Omron CX-Programmer project 新工程 (CX-Programmer 9.73)

# PLC 新PLC1: CQM1H CPU21

## Global symbols (name address type ; comment)
0.00 BOOL  ; 急停
0.01 BOOL  ; 内线
0.02 BOOL  ; 中线
0.03 BOOL  ; 外线
0.04 BOOL  ; 手动上升
0.05 BOOL  ; 手动下降
0.06 BOOL  ; 储坯/进窑
0.07 BOOL  ; 自动/手动
0.08 BOOL  ; 连锁
0.09 BOOL  ; 笼中进
0.10 BOOL  ; 笼中出
0.11 BOOL  ; 新加线开
0.12 BOOL  ; 棒1#光电
0.13 BOOL  ; 棒2#光电
0.14 BOOL  ; 棒3光电
0.15 BOOL  ; 棒8#光电
100.00 BOOL  ; 棒1#快速速
100.01 BOOL  ; 棒1#慢速
100.02 BOOL  ; 内送砖前3#基速
100.03 BOOL  ; 内送砖前3#慢速
100.04 BOOL  ; 中线送砖前3#
100.05 BOOL  ; 中线送砖前3#慢速
100.06 BOOL  ; 外线送砖前3#正转
100.07 BOOL  ; 外线送砖前3#慢速
100.08 BOOL  ; 内线正转
100.09 BOOL  ; 内线慢速
100.10 BOOL  ; 内线反转
100.12 BOOL  ; 中线正转
100.13 BOOL  ; 中线低速
100.14 BOOL  ; 中线反转
101.00 BOOL  ; 外线正转
101.01 BOOL  ; 外线低速
101.02 BOOL  ; 外线反转
101.04 BOOL  ; 棒2#
101.05 BOOL  ; 棒3#
101.06 BOOL  ; 棒4#
101.07 BOOL  ; 棒7#
101.08 BOOL  ; 棒8#
101.09 BOOL  ; 棍9#正转
101.10 BOOL  ; 棍9#反转
101.11 BOOL  ; 棒10#正转
101.12 BOOL  ; 棒10#反转
101.13 BOOL  ; 棒11#正转
101.14 BOOL  ; 棒11#反转
101.15 BOOL  ; 棒12正转（外线）
102.00 BOOL  ; 棒12反转（外线）
102.01 BOOL  ; 1#补棒正转
102.02 BOOL  ; 1#补棒反转
102.03 BOOL  ; 2#补棒正转
102.04 BOOL  ; 2#补棒反转
102.05 BOOL  ; 1#笼棒正转
102.06 BOOL  ; 1#笼棒棒反转
102.07 BOOL  ; 2#笼棒正转
102.08 BOOL  ; 2#笼棒反转
102.09 BOOL  ; 内线送砖前2#
102.10 BOOL  ; 内送砖前1#
102.11 BOOL  ; 内线送砖
102.12 BOOL  ; 内线步进
102.13 BOOL  ; 内线升降
102.14 BOOL  ; 中线送砖前2#
102.15 BOOL  ; 中线送砖前1#
103.00 BOOL  ; 中线送砖
103.01 BOOL  ; 中线步进
103.02 BOOL  ; 中线升降
103.03 BOOL  ; 外线送砖前2#
103.04 BOOL  ; 外线送砖前1#
103.05 BOOL  ; 外线送砖
103.06 BOOL  ; 吊笼上升
103.07 BOOL  ; 吊笼下降
103.08 BOOL  ; 外线步进
103.09 BOOL  ; 外线升降
104.00 BOOL  ; 1线快拉正转
104.01 BOOL  ; 1线快拉反转
104.02 BOOL  ; 1线快拉慢速
104.03 BOOL  ; 1线送砖前4#基速
104.04 BOOL  ; 1线送砖前4#慢速
104.05 BOOL  ; 1线送砖前3#
104.06 BOOL  ; 1线送砖前2#
104.07 BOOL  ; 1线送砖前1#
104.08 BOOL  ; 1线送砖
104.09 BOOL  ; 1线步进
104.10 BOOL  ; 1线升降
104.11 BOOL  ; 棒5
104.12 BOOL  ; 棒6#
10.00 BOOL  ; 砖已离开补棒1#
10.01 BOOL  ; 棒11#放砖
10.02 BOOL  ; 棒11#放砖
10.03 BOOL  ; 棒9#正转
10.05 BOOL  ; 棒9反储启棒10反
10.06 BOOL  ; 棒10反储启棒11反
11.00 BOOL  ; 吊笼自动上升
11.01 BOOL  ; 吊笼手动上升
11.02 BOOL  ; 吊笼上升定位
11.03 BOOL  ; 吊笼自下
11.04 BOOL  ; 吊笼手下
11.05 BOOL  ; 下降定位
11.07 BOOL  ; 补棒1#有砖
12.00 BOOL  ; 棒12#正转
1.00 BOOL  ; 棒10#光电
1.01 BOOL  ; 棒11#光电
1.02 BOOL  ; 补棒光电
1.03 BOOL  ; 补棒对射
1.04 BOOL  ; 吊笼进口对射
1.05 BOOL  ; 斜射
1.06 BOOL  ; 吊笼定长
1.07 BOOL  ; 吊笼定位
1.08 BOOL  ; 上升层定位
1.09 BOOL  ; 下降层限
1.10 BOOL  ; 上限
1.11 BOOL  ; 下限
1.12 BOOL  ; 内送砖前3#光电
1.13 BOOL  ; 内送砖前2#光电
1.14 BOOL  ; 内送砖前1#光电
1.15 BOOL  ; 内线送砖光电
20.00 BOOL  ; 棒7正转
2.00 BOOL  ; 内线定位光电
2.01 BOOL  ; 内线升降接近
2.02 BOOL  ; 内正限
2.03 BOOL  ; 内正慢
2.04 BOOL  ; 内反慢
2.05 BOOL  ; 内反限
2.06 BOOL  ; 中线1#光电
2.07 BOOL  ; 中线送砖前2#光电
2.08 BOOL  ; 中线送砖前1#光电
2.09 BOOL  ; 中线送砖光电
2.10 BOOL  ; 中线定位光电
2.11 BOOL  ; 中线升降接近
2.12 BOOL  ; 中正限
2.13 BOOL  ; 中正慢
2.14 BOOL  ; 中反慢
2.15 BOOL  ; 中反限
3.00 BOOL  ; 外线送砖前3#光电
3.01 BOOL  ; 外线送砖前2#光电
3.02 BOOL  ; 外线送砖前1#光电
3.03 BOOL  ; 外线送砖光电
3.04 BOOL  ; 外线定位光电
3.05 BOOL  ; 外线升降接近
3.06 BOOL  ; 外正限
3.07 BOOL  ; 外正慢
3.08 BOOL  ; 外反慢
3.09 BOOL  ; 外反限
3.14 BOOL  ; 棒4光电
4.00 BOOL  ; 1线快拉正限
4.01 BOOL  ; 1线快拉正慢
4.02 BOOL  ; 1线快拉反限
4.03 BOOL  ; 1线快拉反慢
4.04 BOOL  ; 1线送砖前4#光电
4.05 BOOL  ; 1线送砖前3#光电
4.06 BOOL  ; 1线送砖前2#光电
4.07 BOOL  ; 1线送砖前1#光电
4.08 BOOL  ; 1线送砖光电
4.09 BOOL  ; 1线定位光电
4.10 BOOL  ; 1线升降接近
4.11 BOOL  ; 棒6光电
CNT005 BOOL  ; 棒12#过砖时间
CNT007 BOOL  ; 棒12#放砖时间
CNT008 BOOL  ; 棒11#放砖时间
CNT009 BOOL  ; 棒10#放砖时间
CNT013 BOOL  ; 棒9#放砖时间
CNT015 BOOL  ; 棒9#过砖时间
CNT021 BOOL  ; 棒8放砖时间
CNT022 BOOL  ; 棒7#过砖时间
CNT024 BOOL  ; 棒7#放砖时间
CNT028 BOOL  ; 棒9#反储时间
CNT030 BOOL  ; 棒10#反储时间
CNT032 BOOL  ; 棒11#反储时间
CNT033 BOOL  ; 棒12#反过时间
CNT035 BOOL  ; 棒12#反储时间
CNT038 BOOL  ; 吊笼上升到位
CNT041 BOOL  ; 下降定位
CNT045 BOOL  ; 补棒1#反储定位
CNT051 BOOL  ; 棒11反储时间
CNT053 BOOL  ; 棒10#放砖时间
CNT102 BOOL  ; 棒6放砖时间
CNT103 BOOL  ; 棒5#过砖时间
CNT105 BOOL  ; 棒5#放砖时间
HR0.01 BOOL  ; 内线上升
HR0.02 BOOL  ; 内线快拉正转
HR0.03 BOOL  ; 内线下降
HR0.04 BOOL  ; 内线快拉反转
HR0.05 BOOL  ; 中线上升
HR0.06 BOOL  ; 中线快拉正转
HR0.07 BOOL  ; 中线下降
HR0.08 BOOL  ; 中线快拉反转
HR0.09 BOOL  ; 外线上升
HR0.10 BOOL  ; 外线快拉正转
HR0.11 BOOL  ; 外线下降
HR0.12 BOOL  ; 外线快拉反转
HR0.13 BOOL  ; 笼棒放砖
HR0.14 BOOL  ; 棒12#过砖
HR0.15 BOOL  ; 棒12#放砖
HR10.00 BOOL  ; 棒12放砖至棒11
HR10.01 BOOL  ; 棒11#放砖
HR10.02 BOOL  ; 棒11放砖至棒10
HR10.03 BOOL  ; 棒10#放砖
HR10.04 BOOL  ; 棒9#中线放砖
HR10.05 BOOL  ; 棒9#过砖
HR10.06 BOOL  ; 棒9放砖至棒8
HR10.07 BOOL  ; 棒8#放砖
HR10.08 BOOL  ; 棒7#过砖
HR10.09 BOOL  ; 棒7#放砖
HR10.10 BOOL  ; 中线储坯下降
HR10.11 BOOL  ; 外线储坯下降
HR10.12 BOOL  ; 棒9#反储
HR10.13 BOOL  ; 棒10#反过
HR10.14 BOOL  ; 棒10#反储
HR10.15 BOOL  ; 棒11#反过
HR11.00 BOOL  ; 棒11#反储
HR11.01 BOOL  ; 棒12#反过
HR11.02 BOOL  ; 棒12#反储
HR11.03 BOOL  ; 笼棒反储定长
HR12.00 BOOL  ; 吊笼上升
HR12.01 BOOL  ; 吊笼下降
HR12.02 BOOL  ; 补棒1#反储定长
HR12.04 BOOL  ; 棒10#反储
HR12.05 BOOL  ; 棒10有砖棒11反储
HR12.06 BOOL  ; 棒12放砖至棒11
HR12.07 BOOL  ; 棒10#放砖
HR13.01 BOOL  ; 1线上升
HR13.02 BOOL  ; 1线快拉正转
HR13.03 BOOL  ; 1线下降
HR13.04 BOOL  ; 1线快拉反转
HR13.08 BOOL  ; 棒7放砖至棒6
HR13.09 BOOL  ; 棒6#放砖
HR13.10 BOOL  ; 棒5#过砖
HR13.11 BOOL  ; 棒5#放砖
TIM000 BOOL  ; 棒1#无砖
TIM001 BOOL  ; 内线快拉正转后
TIM002 BOOL  ; 中线快拉正转
TIM003 BOOL  ; 外线快拉正转
TIM004 BOOL  ; 放砖条件
TIM006 BOOL  ; 外线下降
TIM010 BOOL  ; 棒11砖定位
TIM011 BOOL  ; 棒10砖定位
TIM012 BOOL  ; 中线下降
TIM020 BOOL  ; 棒8#砖定位
TIM023 BOOL  ; 内线下降
TIM025 BOOL  ; 中线储坯下降条件
TIM026 BOOL  ; 外线储坯下降条件
TIM027 BOOL  ; 中线储坯下降
TIM029 BOOL  ; 棒10#反过定位
TIM031 BOOL  ; 棒11#反过定位
TIM034 BOOL  ; 外线储坯下降
TIM036 BOOL  ; 吊笼上升条件
TIM037 BOOL  ; 上升层定位
TIM039 BOOL  ; 吊笼下降条件
TIM040 BOOL  ; 下降层定位
TIM042 BOOL  ; 棒10#放砖条件
TIM043 BOOL  ; 棒11放砖条件
TIM050 BOOL  ; 定位
TIM052 BOOL  ; 棒11砖定位
TIM055 BOOL  ; 棒10#放砖条件
TIM100 BOOL  ; 1线快拉正转后
TIM101 BOOL  ; 棒6#砖定位
TIM104 BOOL  ; 1线下降

## Program 新程序1 (no task)
; 程序使用CX-Programmer 9.75编写，PLC型号为CQM1H CPU21。程序实现了陶瓷厂储坯器系统的控制系统，通过输送带控制坯料输送、升降机调整坯料位置和吊笼实现坯料存储。操作人员通过自动/手动开关选择运行模式，自动和手动模式不能同时启用。 / 设备情况：输送带、升降机、吊笼、急停按钮、连锁开关、光电传感器、限位开关和接近开关等。 / 操作员可以通过自动/手动开关选择运行模式，在自动模式下，运转准备信号和插头连接确认信号确认后点亮自动运转指示灯。若插头连接确认信号为假，检测暂停，自动运转指示灯不点亮，直到插头重新连接。检测流程由放水电磁阀和电机运转继电器控制，通过压力到达信号确保压力达标。 / 输送带控制方面，内线启动按钮启动内线正转输出，需内线送砖光电持续为真。内线输送启动前，确认内线送砖光电信号。中线启动按钮控制中线正转输出，需中线送砖光电信号正常；中线输送启动前，检测中线送砖光电状态。外线启动按钮控制外线正转输出，需外线送砖光电信号有效；外线输送启动前，确保外线送砖光电有效。内线升降输出运行时，需内线升降接近为真以确认位置；内线升降启动时，检查内线升降接近是否到位；内线升降完成时，记录运行状态；内线正转输出此时停止，避免部件掉落。 / 吊笼由吊笼上升输出和吊笼下降输出控制，在自动模式下由运转准备信号和上限信号触发上升，手动模式下由手动上升按钮和手动下降按钮操作。吊笼停止前，检测吊笼进口对射是否正常。吊笼运行时，吊笼进口对射必须为真以检测障碍物，否则停止运行，避免撞击。吊笼定位控制移动，上限信号和下限信号限制移动范围。 / 安全方面，急停按钮按下时，内线正转输出、吊笼上升输出等所有输出立即停止，确保人员和设备安全；系统启动前，检测急停按钮是否复位。若连锁开关为假，内线正转输出、电机运转继电器等主要输出停止运行，防止不安全状态下的操作；输送开始前，确认连锁开关已闭合。不良状态下，操作员按下不良解除按钮可复位系统，恢复初始状态。 / 内线正转输出运行时需持续检测内线送砖光电，中线正转输出需持续检测中线送砖光电，外线正转输出需持续检测外线送砖光电，否则停止运行以防部件堆积。 / 内线升降输出运行时需持续检测内线升降接近，中线升降输出需持续检测中线升降接近，外线升降输出需持续检测外线升降接近，以确保位置正常；中线升降前，验证中线升降接近信号；外线升降开始前，确认外线升降接近正常。

### Section 段1

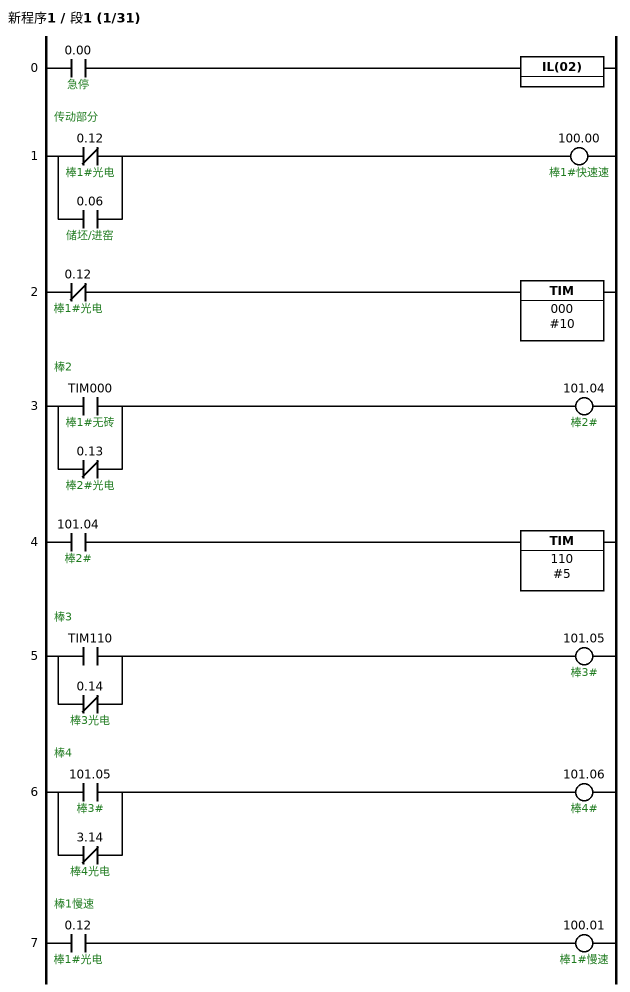
; rung 0
LD 0.00  ; 急停
IL(02)
; rung 1: 传动部分
LDNOT 0.12  ; 棒1#光电
OR 0.06  ; 储坯/进窑
OUT 100.00  ; 棒1#快速速
; rung 2
LDNOT 0.12  ; 棒1#光电
TIM 000 #10
; rung 3: 棒2
LD TIM000  ; 棒1#无砖
ORNOT 0.13  ; 棒2#光电
OUT 101.04  ; 棒2#
; rung 4
LD 101.04  ; 棒2#
TIM 110 #5
; rung 5: 棒3
LD TIM110
ORNOT 0.14  ; 棒3光电
OUT 101.05  ; 棒3#
; rung 6: 棒4
LD 101.05  ; 棒3#
ORNOT 3.14  ; 棒4光电
OUT 101.06  ; 棒4#
; rung 7: 棒1慢速
LD 0.12  ; 棒1#光电
OUT 100.01  ; 棒1#慢速

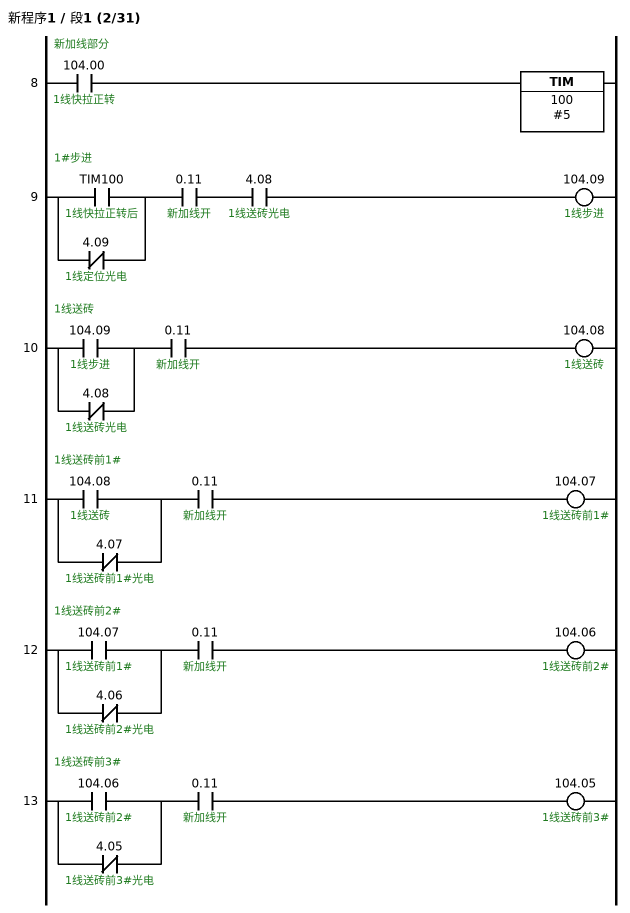
; rung 8: 新加线部分
LD 104.00  ; 1线快拉正转
TIM 100 #5
; rung 9: 1#步进
LD TIM100  ; 1线快拉正转后
ORNOT 4.09  ; 1线定位光电
AND 0.11  ; 新加线开
AND 4.08  ; 1线送砖光电
OUT 104.09  ; 1线步进
; rung 10: 1线送砖
LD 104.09  ; 1线步进
ORNOT 4.08  ; 1线送砖光电
AND 0.11  ; 新加线开
OUT 104.08  ; 1线送砖
; rung 11: 1线送砖前1#
LD 104.08  ; 1线送砖
ORNOT 4.07  ; 1线送砖前1#光电
AND 0.11  ; 新加线开
OUT 104.07  ; 1线送砖前1#
; rung 12: 1线送砖前2#
LD 104.07  ; 1线送砖前1#
ORNOT 4.06  ; 1线送砖前2#光电
AND 0.11  ; 新加线开
OUT 104.06  ; 1线送砖前2#
; rung 13: 1线送砖前3#
LD 104.06  ; 1线送砖前2#
ORNOT 4.05  ; 1线送砖前3#光电
AND 0.11  ; 新加线开
OUT 104.05  ; 1线送砖前3#

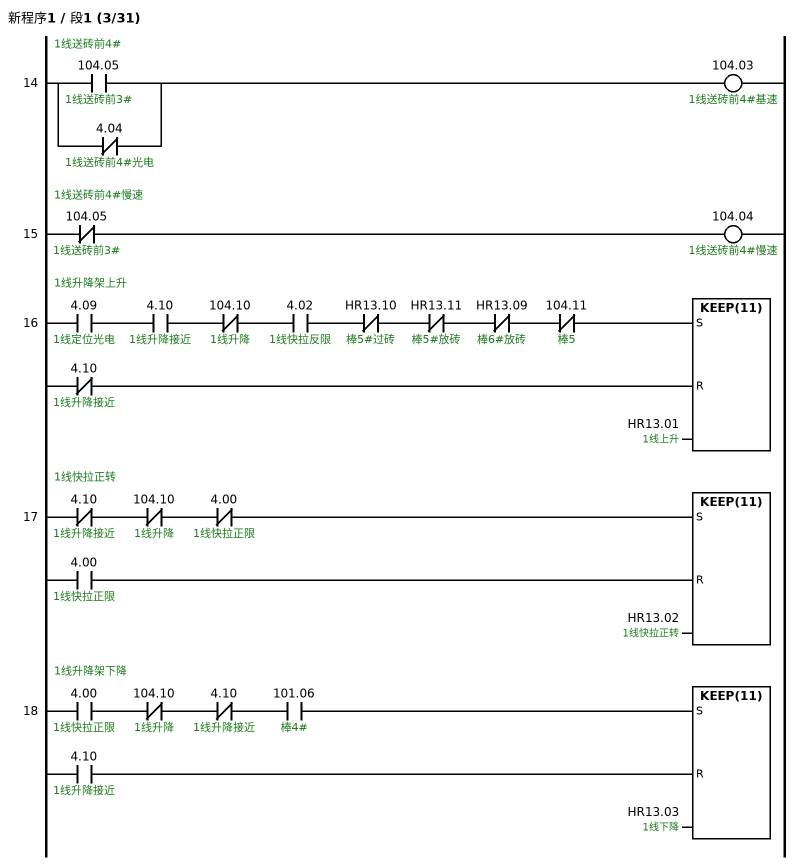
; rung 14: 1线送砖前4#
LD 104.05  ; 1线送砖前3#
ORNOT 4.04  ; 1线送砖前4#光电
OUT 104.03  ; 1线送砖前4#基速
; rung 15: 1线送砖前4#慢速
LDNOT 104.05  ; 1线送砖前3#
OUT 104.04  ; 1线送砖前4#慢速
; rung 16: 1线升降架上升
LD 4.09  ; 1线定位光电
AND 4.10  ; 1线升降接近
ANDNOT 104.10  ; 1线升降
AND 4.02  ; 1线快拉反限
ANDNOT HR13.10  ; 棒5#过砖
ANDNOT HR13.11  ; 棒5#放砖
ANDNOT HR13.09  ; 棒6#放砖
ANDNOT 104.11  ; 棒5
LDNOT 4.10  ; 1线升降接近
KEEP(11) HR13.01  ; 1线上升
; rung 17: 1线快拉正转
LDNOT 4.10  ; 1线升降接近
ANDNOT 104.10  ; 1线升降
ANDNOT 4.00  ; 1线快拉正限
LD 4.00  ; 1线快拉正限
KEEP(11) HR13.02  ; 1线快拉正转
; rung 18: 1线升降架下降
LD 4.00  ; 1线快拉正限
ANDNOT 104.10  ; 1线升降
ANDNOT 4.10  ; 1线升降接近
AND 101.06  ; 棒4#
LD 4.10  ; 1线升降接近
KEEP(11) HR13.03  ; 1线下降

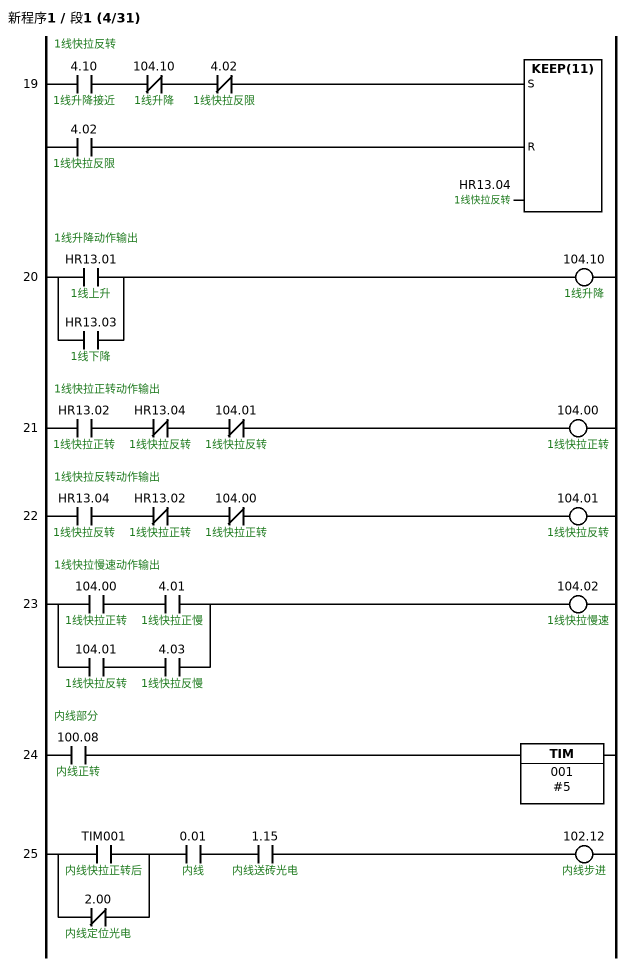
; rung 19: 1线快拉反转
LD 4.10  ; 1线升降接近
ANDNOT 104.10  ; 1线升降
ANDNOT 4.02  ; 1线快拉反限
LD 4.02  ; 1线快拉反限
KEEP(11) HR13.04  ; 1线快拉反转
; rung 20: 1线升降动作输出
LD HR13.01  ; 1线上升
OR HR13.03  ; 1线下降
OUT 104.10  ; 1线升降
; rung 21: 1线快拉正转动作输出
LD HR13.02  ; 1线快拉正转
ANDNOT HR13.04  ; 1线快拉反转
ANDNOT 104.01  ; 1线快拉反转
OUT 104.00  ; 1线快拉正转
; rung 22: 1线快拉反转动作输出
LD HR13.04  ; 1线快拉反转
ANDNOT HR13.02  ; 1线快拉正转
ANDNOT 104.00  ; 1线快拉正转
OUT 104.01  ; 1线快拉反转
; rung 23: 1线快拉慢速动作输出
LD 104.00  ; 1线快拉正转
AND 4.01  ; 1线快拉正慢
LD 104.01  ; 1线快拉反转
AND 4.03  ; 1线快拉反慢
ORLD
OUT 104.02  ; 1线快拉慢速
; rung 24: 内线部分
LD 100.08  ; 内线正转
TIM 001 #5
; rung 25
LD TIM001  ; 内线快拉正转后
ORNOT 2.00  ; 内线定位光电
AND 0.01  ; 内线
AND 1.15  ; 内线送砖光电
OUT 102.12  ; 内线步进

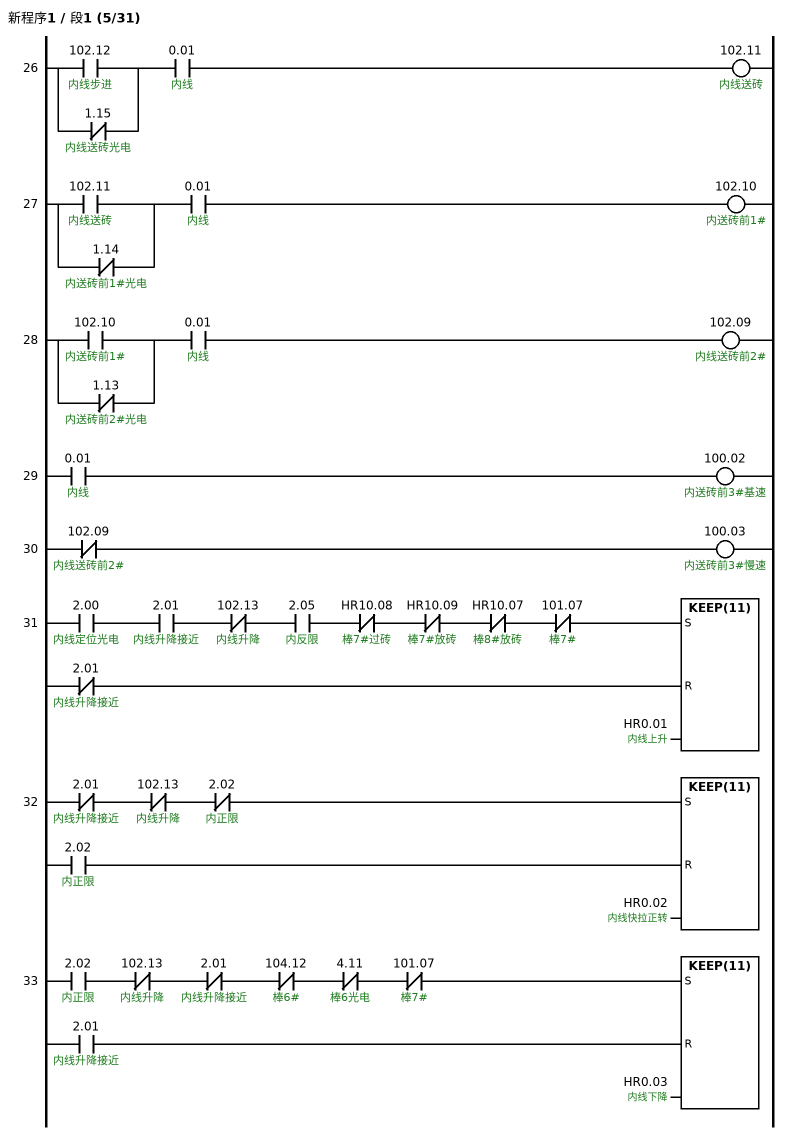
; rung 26
LD 102.12  ; 内线步进
ORNOT 1.15  ; 内线送砖光电
AND 0.01  ; 内线
OUT 102.11  ; 内线送砖
; rung 27
LD 102.11  ; 内线送砖
ORNOT 1.14  ; 内送砖前1#光电
AND 0.01  ; 内线
OUT 102.10  ; 内送砖前1#
; rung 28
LD 102.10  ; 内送砖前1#
ORNOT 1.13  ; 内送砖前2#光电
AND 0.01  ; 内线
OUT 102.09  ; 内线送砖前2#
; rung 29
LD 0.01  ; 内线
OUT 100.02  ; 内送砖前3#基速
; rung 30
LDNOT 102.09  ; 内线送砖前2#
OUT 100.03  ; 内送砖前3#慢速
; rung 31
LD 2.00  ; 内线定位光电
AND 2.01  ; 内线升降接近
ANDNOT 102.13  ; 内线升降
AND 2.05  ; 内反限
ANDNOT HR10.08  ; 棒7#过砖
ANDNOT HR10.09  ; 棒7#放砖
ANDNOT HR10.07  ; 棒8#放砖
ANDNOT 101.07  ; 棒7#
LDNOT 2.01  ; 内线升降接近
KEEP(11) HR0.01  ; 内线上升
; rung 32
LDNOT 2.01  ; 内线升降接近
ANDNOT 102.13  ; 内线升降
ANDNOT 2.02  ; 内正限
LD 2.02  ; 内正限
KEEP(11) HR0.02  ; 内线快拉正转
; rung 33
LD 2.02  ; 内正限
ANDNOT 102.13  ; 内线升降
ANDNOT 2.01  ; 内线升降接近
ANDNOT 104.12  ; 棒6#
ANDNOT 4.11  ; 棒6光电
ANDNOT 101.07  ; 棒7#
LD 2.01  ; 内线升降接近
KEEP(11) HR0.03  ; 内线下降

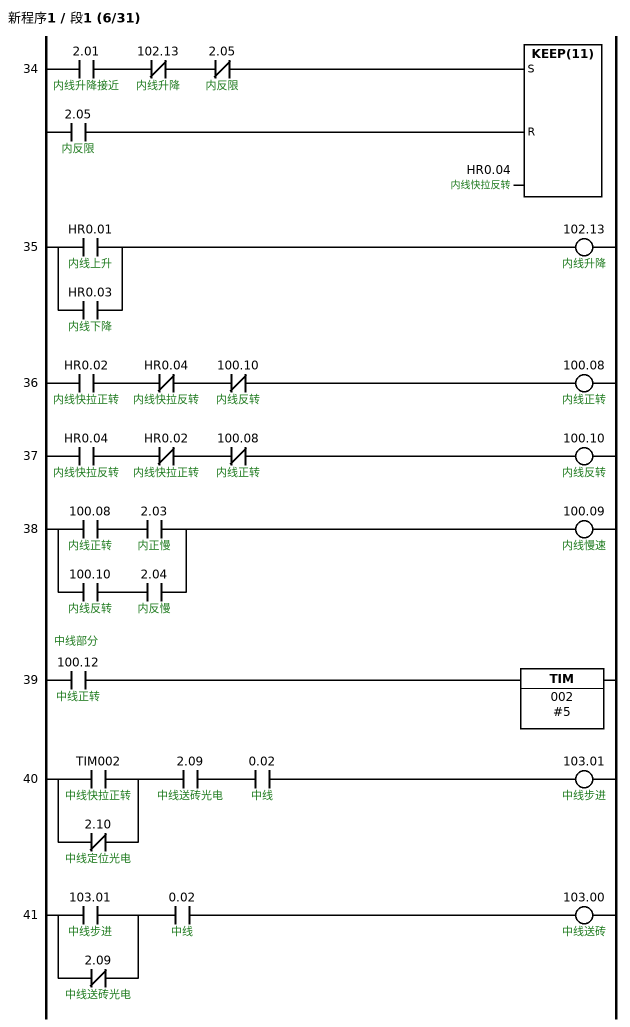
; rung 34
LD 2.01  ; 内线升降接近
ANDNOT 102.13  ; 内线升降
ANDNOT 2.05  ; 内反限
LD 2.05  ; 内反限
KEEP(11) HR0.04  ; 内线快拉反转
; rung 35
LD HR0.01  ; 内线上升
OR HR0.03  ; 内线下降
OUT 102.13  ; 内线升降
; rung 36
LD HR0.02  ; 内线快拉正转
ANDNOT HR0.04  ; 内线快拉反转
ANDNOT 100.10  ; 内线反转
OUT 100.08  ; 内线正转
; rung 37
LD HR0.04  ; 内线快拉反转
ANDNOT HR0.02  ; 内线快拉正转
ANDNOT 100.08  ; 内线正转
OUT 100.10  ; 内线反转
; rung 38
LD 100.08  ; 内线正转
AND 2.03  ; 内正慢
LD 100.10  ; 内线反转
AND 2.04  ; 内反慢
ORLD
OUT 100.09  ; 内线慢速
; rung 39: 中线部分
LD 100.12  ; 中线正转
TIM 002 #5
; rung 40
LD TIM002  ; 中线快拉正转
ORNOT 2.10  ; 中线定位光电
AND 2.09  ; 中线送砖光电
AND 0.02  ; 中线
OUT 103.01  ; 中线步进
; rung 41
LD 103.01  ; 中线步进
ORNOT 2.09  ; 中线送砖光电
AND 0.02  ; 中线
OUT 103.00  ; 中线送砖

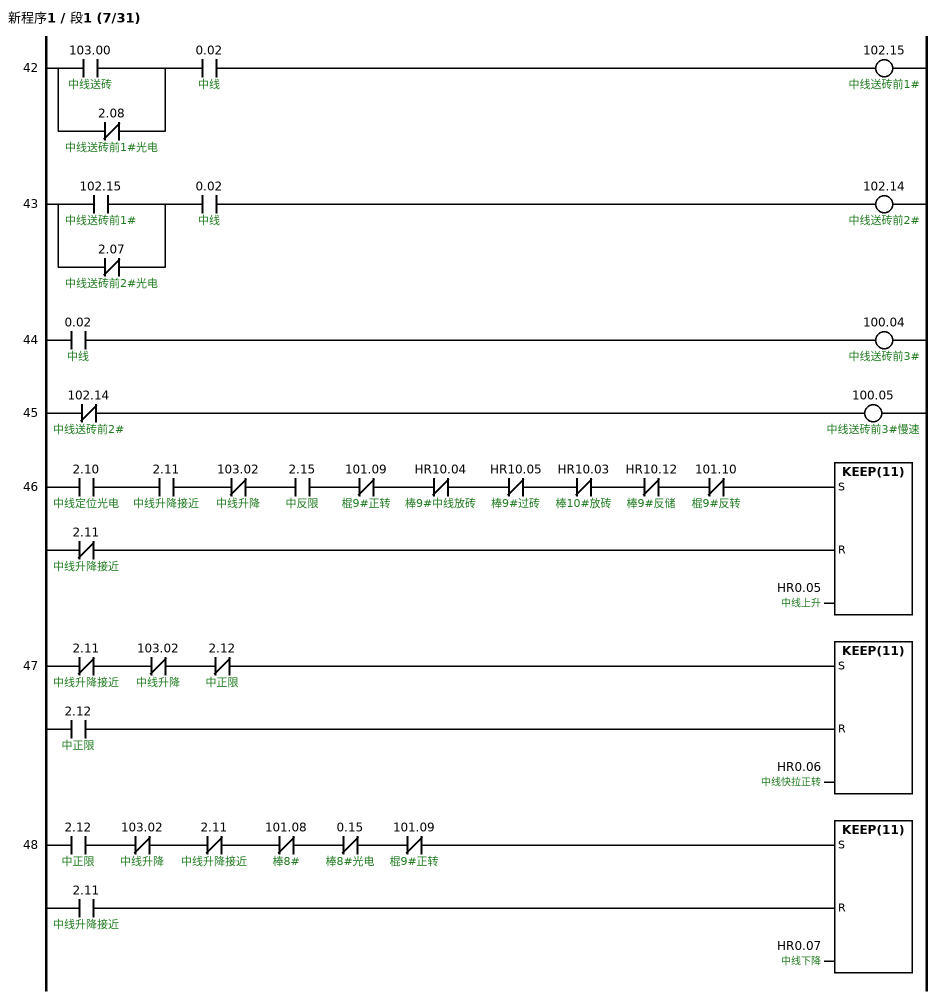
; rung 42
LD 103.00  ; 中线送砖
ORNOT 2.08  ; 中线送砖前1#光电
AND 0.02  ; 中线
OUT 102.15  ; 中线送砖前1#
; rung 43
LD 102.15  ; 中线送砖前1#
ORNOT 2.07  ; 中线送砖前2#光电
AND 0.02  ; 中线
OUT 102.14  ; 中线送砖前2#
; rung 44
LD 0.02  ; 中线
OUT 100.04  ; 中线送砖前3#
; rung 45
LDNOT 102.14  ; 中线送砖前2#
OUT 100.05  ; 中线送砖前3#慢速
; rung 46
LD 2.10  ; 中线定位光电
AND 2.11  ; 中线升降接近
ANDNOT 103.02  ; 中线升降
AND 2.15  ; 中反限
ANDNOT 101.09  ; 棍9#正转
ANDNOT HR10.04  ; 棒9#中线放砖
ANDNOT HR10.05  ; 棒9#过砖
ANDNOT HR10.03  ; 棒10#放砖
ANDNOT HR10.12  ; 棒9#反储
ANDNOT 101.10  ; 棍9#反转
LDNOT 2.11  ; 中线升降接近
KEEP(11) HR0.05  ; 中线上升
; rung 47
LDNOT 2.11  ; 中线升降接近
ANDNOT 103.02  ; 中线升降
ANDNOT 2.12  ; 中正限
LD 2.12  ; 中正限
KEEP(11) HR0.06  ; 中线快拉正转
; rung 48
LD 2.12  ; 中正限
ANDNOT 103.02  ; 中线升降
ANDNOT 2.11  ; 中线升降接近
ANDNOT 101.08  ; 棒8#
ANDNOT 0.15  ; 棒8#光电
ANDNOT 101.09  ; 棍9#正转
LD 2.11  ; 中线升降接近
KEEP(11) HR0.07  ; 中线下降

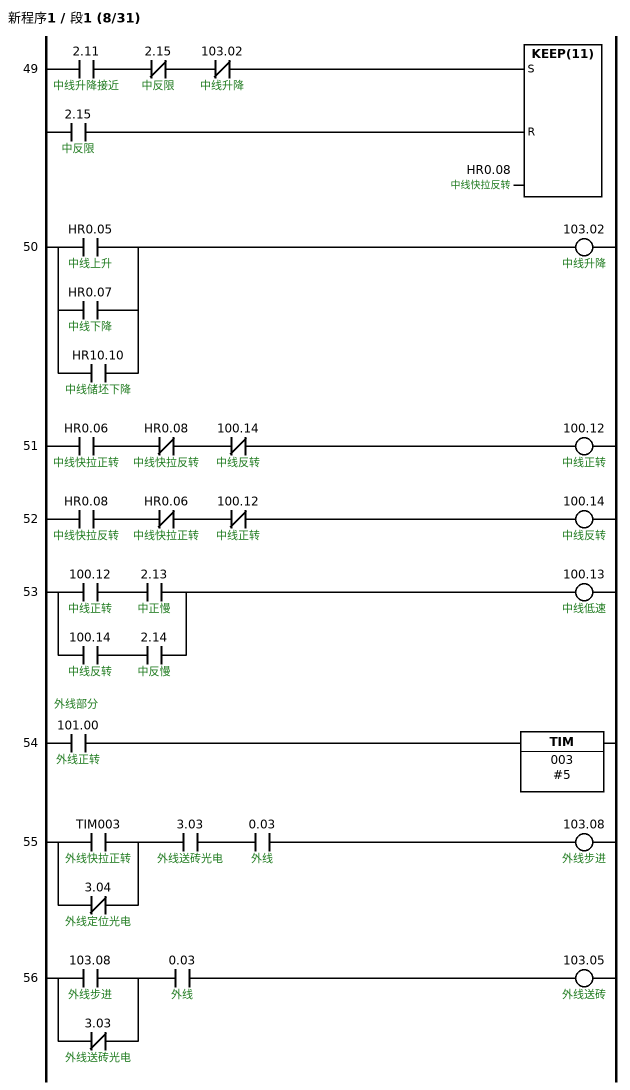
; rung 49
LD 2.11  ; 中线升降接近
ANDNOT 2.15  ; 中反限
ANDNOT 103.02  ; 中线升降
LD 2.15  ; 中反限
KEEP(11) HR0.08  ; 中线快拉反转
; rung 50
LD HR0.05  ; 中线上升
OR HR0.07  ; 中线下降
OR HR10.10  ; 中线储坯下降
OUT 103.02  ; 中线升降
; rung 51
LD HR0.06  ; 中线快拉正转
ANDNOT HR0.08  ; 中线快拉反转
ANDNOT 100.14  ; 中线反转
OUT 100.12  ; 中线正转
; rung 52
LD HR0.08  ; 中线快拉反转
ANDNOT HR0.06  ; 中线快拉正转
ANDNOT 100.12  ; 中线正转
OUT 100.14  ; 中线反转
; rung 53
LD 100.12  ; 中线正转
AND 2.13  ; 中正慢
LD 100.14  ; 中线反转
AND 2.14  ; 中反慢
ORLD
OUT 100.13  ; 中线低速
; rung 54: 外线部分
LD 101.00  ; 外线正转
TIM 003 #5
; rung 55
LD TIM003  ; 外线快拉正转
ORNOT 3.04  ; 外线定位光电
AND 3.03  ; 外线送砖光电
AND 0.03  ; 外线
OUT 103.08  ; 外线步进
; rung 56
LD 103.08  ; 外线步进
ORNOT 3.03  ; 外线送砖光电
AND 0.03  ; 外线
OUT 103.05  ; 外线送砖

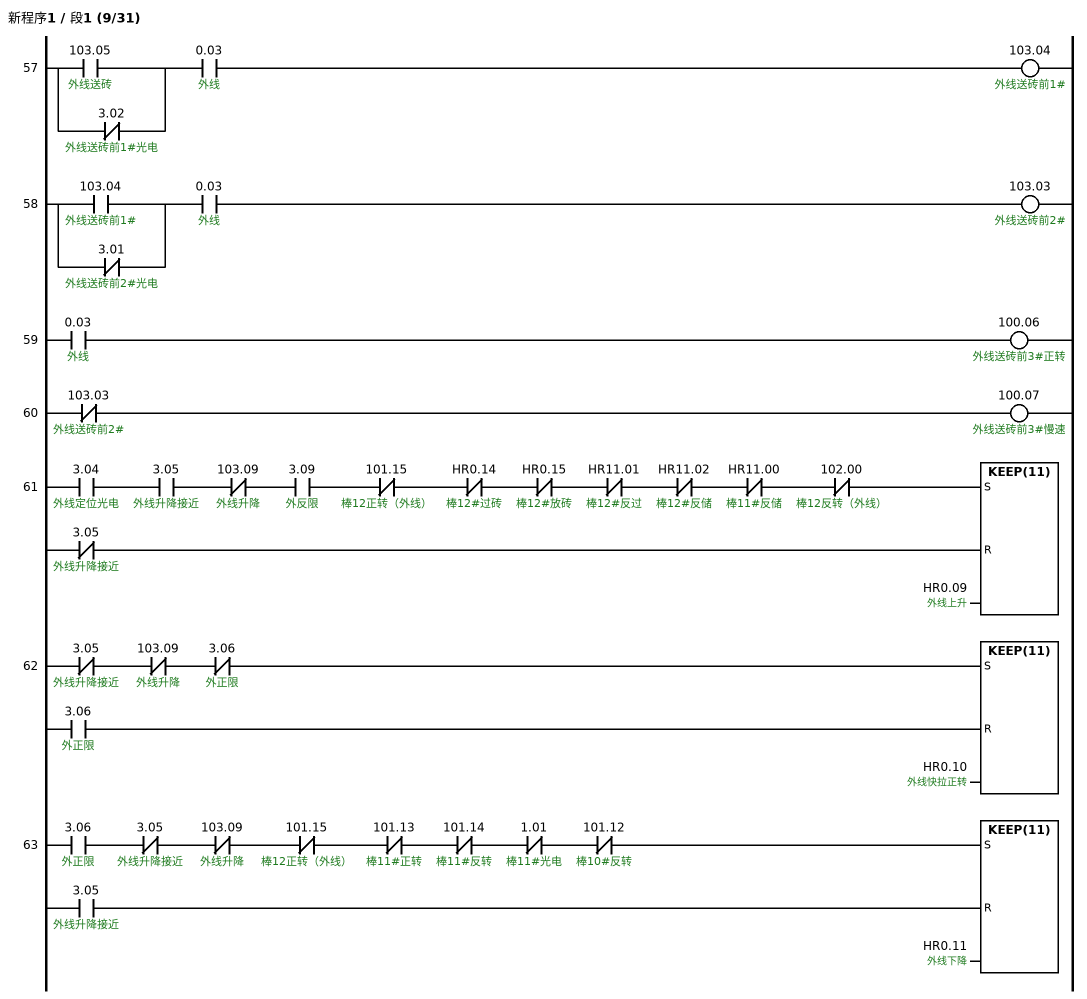
; rung 57
LD 103.05  ; 外线送砖
ORNOT 3.02  ; 外线送砖前1#光电
AND 0.03  ; 外线
OUT 103.04  ; 外线送砖前1#
; rung 58
LD 103.04  ; 外线送砖前1#
ORNOT 3.01  ; 外线送砖前2#光电
AND 0.03  ; 外线
OUT 103.03  ; 外线送砖前2#
; rung 59
LD 0.03  ; 外线
OUT 100.06  ; 外线送砖前3#正转
; rung 60
LDNOT 103.03  ; 外线送砖前2#
OUT 100.07  ; 外线送砖前3#慢速
; rung 61
LD 3.04  ; 外线定位光电
AND 3.05  ; 外线升降接近
ANDNOT 103.09  ; 外线升降
AND 3.09  ; 外反限
ANDNOT 101.15  ; 棒12正转（外线）
ANDNOT HR0.14  ; 棒12#过砖
ANDNOT HR0.15  ; 棒12#放砖
ANDNOT HR11.01  ; 棒12#反过
ANDNOT HR11.02  ; 棒12#反储
ANDNOT HR11.00  ; 棒11#反储
ANDNOT 102.00  ; 棒12反转（外线）
LDNOT 3.05  ; 外线升降接近
KEEP(11) HR0.09  ; 外线上升
; rung 62
LDNOT 3.05  ; 外线升降接近
ANDNOT 103.09  ; 外线升降
ANDNOT 3.06  ; 外正限
LD 3.06  ; 外正限
KEEP(11) HR0.10  ; 外线快拉正转
; rung 63
LD 3.06  ; 外正限
ANDNOT 3.05  ; 外线升降接近
ANDNOT 103.09  ; 外线升降
ANDNOT 101.15  ; 棒12正转（外线）
ANDNOT 101.13  ; 棒11#正转
ANDNOT 101.14  ; 棒11#反转
ANDNOT 1.01  ; 棒11#光电
ANDNOT 101.12  ; 棒10#反转
LD 3.05  ; 外线升降接近
KEEP(11) HR0.11  ; 外线下降

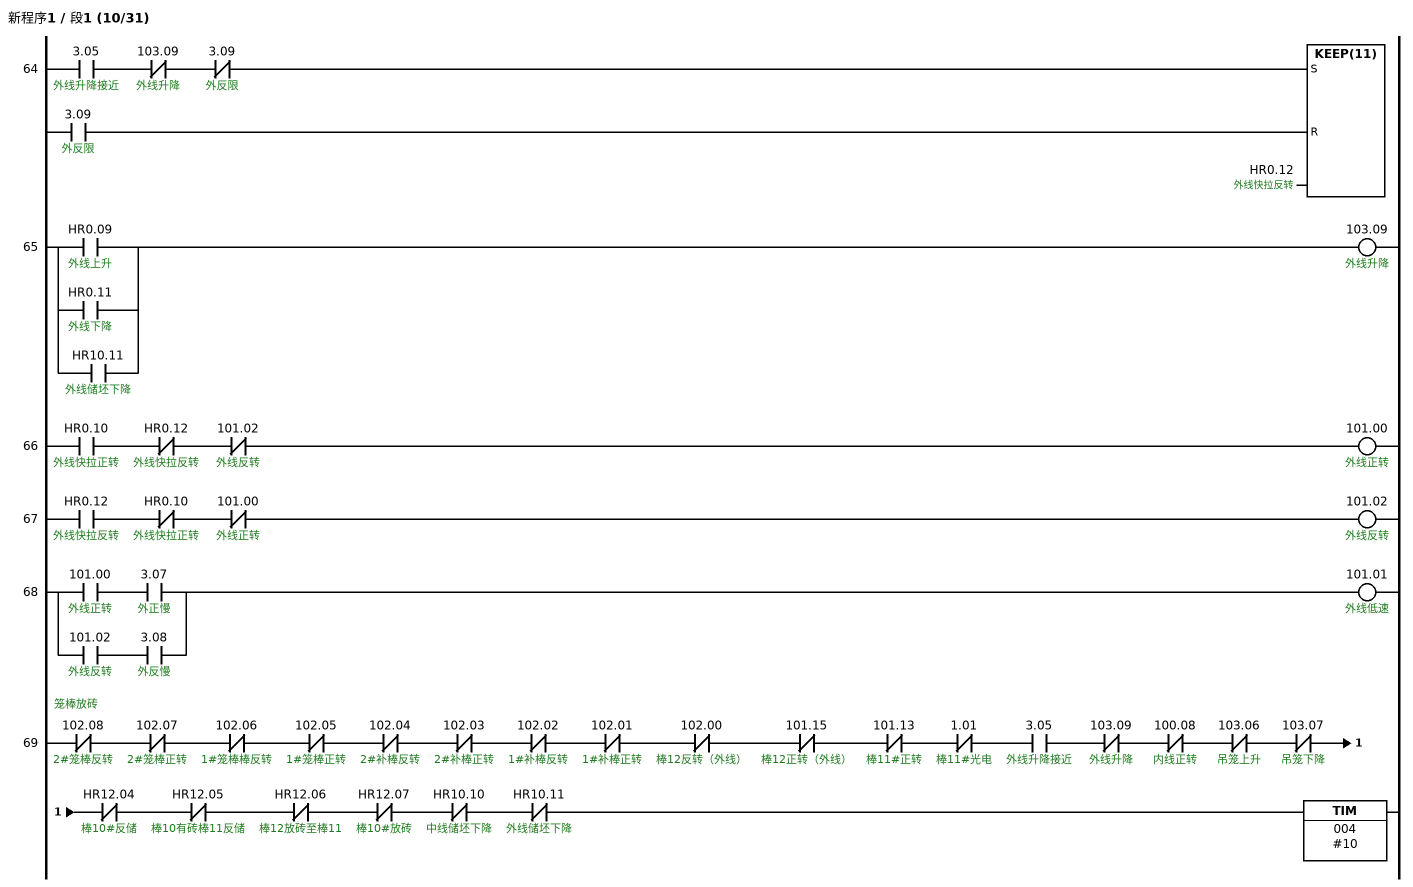
; rung 64
LD 3.05  ; 外线升降接近
ANDNOT 103.09  ; 外线升降
ANDNOT 3.09  ; 外反限
LD 3.09  ; 外反限
KEEP(11) HR0.12  ; 外线快拉反转
; rung 65
LD HR0.09  ; 外线上升
OR HR0.11  ; 外线下降
OR HR10.11  ; 外线储坯下降
OUT 103.09  ; 外线升降
; rung 66
LD HR0.10  ; 外线快拉正转
ANDNOT HR0.12  ; 外线快拉反转
ANDNOT 101.02  ; 外线反转
OUT 101.00  ; 外线正转
; rung 67
LD HR0.12  ; 外线快拉反转
ANDNOT HR0.10  ; 外线快拉正转
ANDNOT 101.00  ; 外线正转
OUT 101.02  ; 外线反转
; rung 68
LD 101.00  ; 外线正转
AND 3.07  ; 外正慢
LD 101.02  ; 外线反转
AND 3.08  ; 外反慢
ORLD
OUT 101.01  ; 外线低速
; rung 69: 笼棒放砖
LDNOT 102.08  ; 2#笼棒反转
ANDNOT 102.07  ; 2#笼棒正转
ANDNOT 102.06  ; 1#笼棒棒反转
ANDNOT 102.05  ; 1#笼棒正转
ANDNOT 102.04  ; 2#补棒反转
ANDNOT 102.03  ; 2#补棒正转
ANDNOT 102.02  ; 1#补棒反转
ANDNOT 102.01  ; 1#补棒正转
ANDNOT 102.00  ; 棒12反转（外线）
ANDNOT 101.15  ; 棒12正转（外线）
ANDNOT 101.13  ; 棒11#正转
ANDNOT 1.01  ; 棒11#光电
AND 3.05  ; 外线升降接近
ANDNOT 103.09  ; 外线升降
ANDNOT 100.08  ; 内线正转
ANDNOT 103.06  ; 吊笼上升
ANDNOT 103.07  ; 吊笼下降
ANDNOT HR12.04  ; 棒10#反储
ANDNOT HR12.05  ; 棒10有砖棒11反储
ANDNOT HR12.06  ; 棒12放砖至棒11
ANDNOT HR12.07  ; 棒10#放砖
ANDNOT HR10.10  ; 中线储坯下降
ANDNOT HR10.11  ; 外线储坯下降
TIM 004 #10

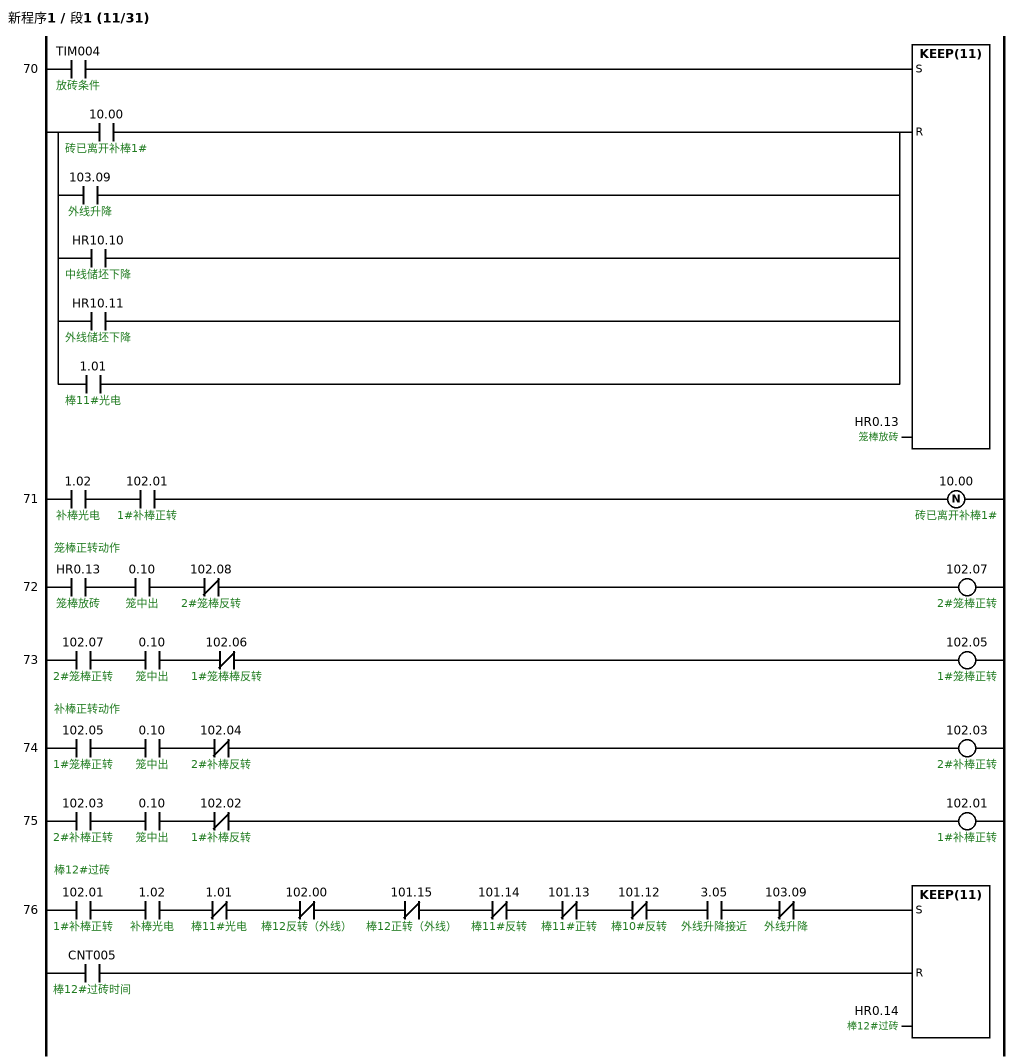
; rung 70
LD TIM004  ; 放砖条件
LD 10.00  ; 砖已离开补棒1#
OR 103.09  ; 外线升降
OR HR10.10  ; 中线储坯下降
OR HR10.11  ; 外线储坯下降
OR 1.01  ; 棒11#光电
KEEP(11) HR0.13  ; 笼棒放砖
; rung 71
LD 1.02  ; 补棒光电
AND 102.01  ; 1#补棒正转
DIFD(14) 10.00  ; 砖已离开补棒1#
; rung 72: 笼棒正转动作
LD HR0.13  ; 笼棒放砖
AND 0.10  ; 笼中出
ANDNOT 102.08  ; 2#笼棒反转
OUT 102.07  ; 2#笼棒正转
; rung 73
LD 102.07  ; 2#笼棒正转
AND 0.10  ; 笼中出
ANDNOT 102.06  ; 1#笼棒棒反转
OUT 102.05  ; 1#笼棒正转
; rung 74: 补棒正转动作
LD 102.05  ; 1#笼棒正转
AND 0.10  ; 笼中出
ANDNOT 102.04  ; 2#补棒反转
OUT 102.03  ; 2#补棒正转
; rung 75
LD 102.03  ; 2#补棒正转
AND 0.10  ; 笼中出
ANDNOT 102.02  ; 1#补棒反转
OUT 102.01  ; 1#补棒正转
; rung 76: 棒12#过砖
LD 102.01  ; 1#补棒正转
AND 1.02  ; 补棒光电
ANDNOT 1.01  ; 棒11#光电
ANDNOT 102.00  ; 棒12反转（外线）
ANDNOT 101.15  ; 棒12正转（外线）
ANDNOT 101.14  ; 棒11#反转
ANDNOT 101.13  ; 棒11#正转
ANDNOT 101.12  ; 棒10#反转
AND 3.05  ; 外线升降接近
ANDNOT 103.09  ; 外线升降
LD CNT005  ; 棒12#过砖时间
KEEP(11) HR0.14  ; 棒12#过砖

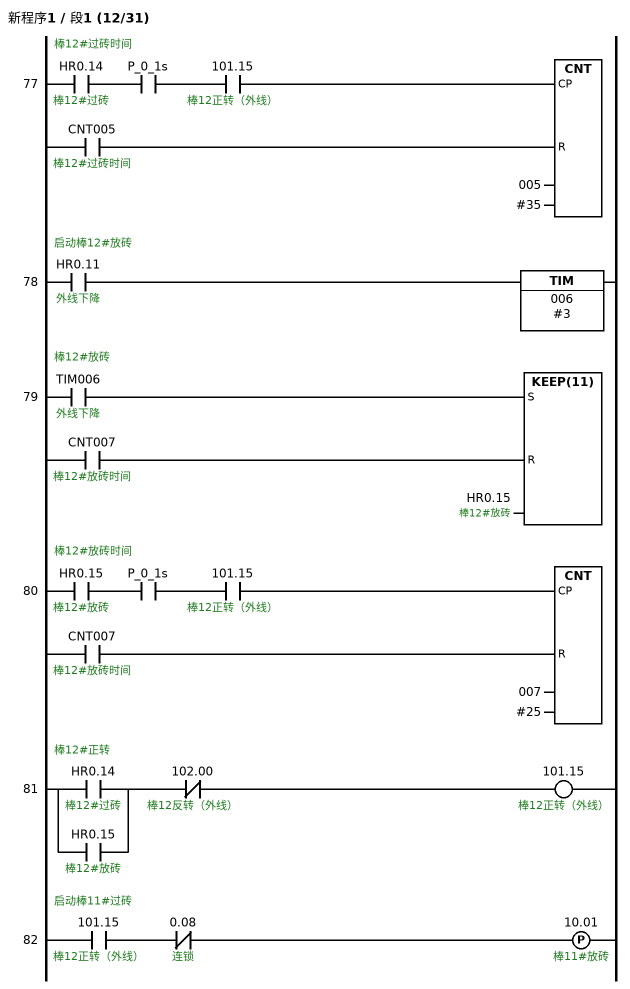
; rung 77: 棒12#过砖时间
LD HR0.14  ; 棒12#过砖
AND P_0_1s
AND 101.15  ; 棒12正转（外线）
LD CNT005  ; 棒12#过砖时间
CNT 005 #35
; rung 78: 启动棒12#放砖
LD HR0.11  ; 外线下降
TIM 006 #3
; rung 79: 棒12#放砖
LD TIM006  ; 外线下降
LD CNT007  ; 棒12#放砖时间
KEEP(11) HR0.15  ; 棒12#放砖
; rung 80: 棒12#放砖时间
LD HR0.15  ; 棒12#放砖
AND P_0_1s
AND 101.15  ; 棒12正转（外线）
LD CNT007  ; 棒12#放砖时间
CNT 007 #25
; rung 81: 棒12#正转
LD HR0.14  ; 棒12#过砖
OR HR0.15  ; 棒12#放砖
ANDNOT 102.00  ; 棒12反转（外线）
OUT 101.15  ; 棒12正转（外线）
; rung 82: 启动棒11#过砖
LD 101.15  ; 棒12正转（外线）
ANDNOT 0.08  ; 连锁
DIFU(13) 10.01  ; 棒11#放砖

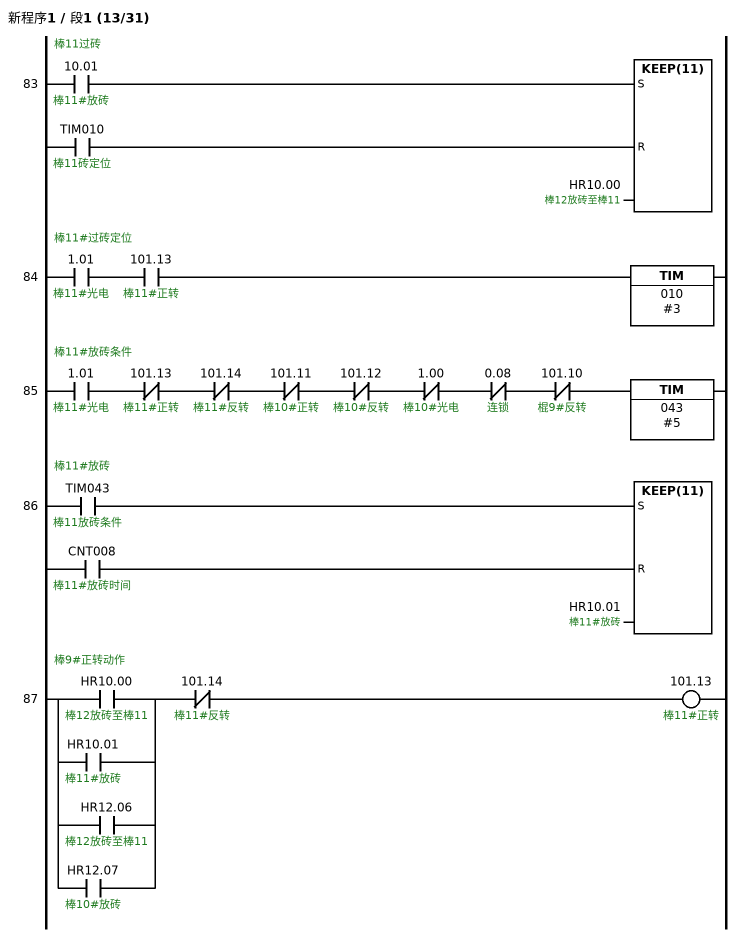
; rung 83: 棒11过砖
LD 10.01  ; 棒11#放砖
LD TIM010  ; 棒11砖定位
KEEP(11) HR10.00  ; 棒12放砖至棒11
; rung 84: 棒11#过砖定位
LD 1.01  ; 棒11#光电
AND 101.13  ; 棒11#正转
TIM 010 #3
; rung 85: 棒11#放砖条件
LD 1.01  ; 棒11#光电
ANDNOT 101.13  ; 棒11#正转
ANDNOT 101.14  ; 棒11#反转
ANDNOT 101.11  ; 棒10#正转
ANDNOT 101.12  ; 棒10#反转
ANDNOT 1.00  ; 棒10#光电
ANDNOT 0.08  ; 连锁
ANDNOT 101.10  ; 棍9#反转
TIM 043 #5
; rung 86: 棒11#放砖
LD TIM043  ; 棒11放砖条件
LD CNT008  ; 棒11#放砖时间
KEEP(11) HR10.01  ; 棒11#放砖
; rung 87: 棒9#正转动作
LD HR10.00  ; 棒12放砖至棒11
OR HR10.01  ; 棒11#放砖
OR HR12.06  ; 棒12放砖至棒11
OR HR12.07  ; 棒10#放砖
ANDNOT 101.14  ; 棒11#反转
OUT 101.13  ; 棒11#正转

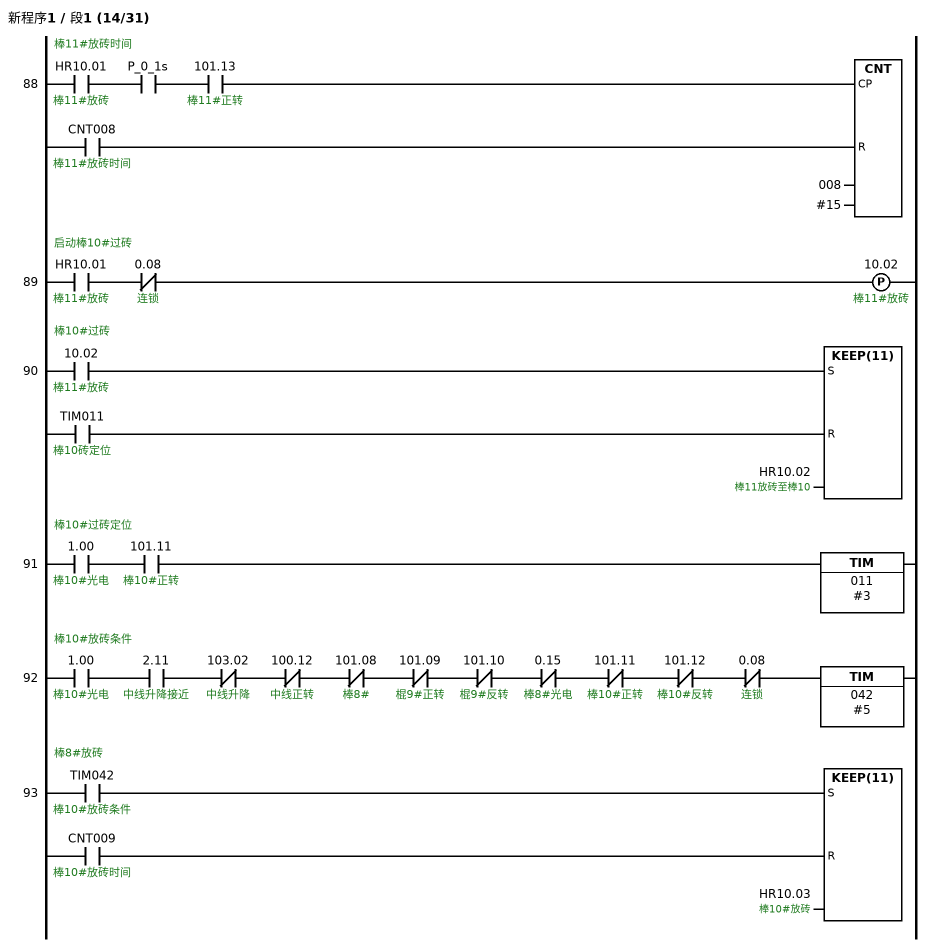
; rung 88: 棒11#放砖时间
LD HR10.01  ; 棒11#放砖
AND P_0_1s
AND 101.13  ; 棒11#正转
LD CNT008  ; 棒11#放砖时间
CNT 008 #15
; rung 89: 启动棒10#过砖
LD HR10.01  ; 棒11#放砖
ANDNOT 0.08  ; 连锁
DIFU(13) 10.02  ; 棒11#放砖
; rung 90: 棒10#过砖
LD 10.02  ; 棒11#放砖
LD TIM011  ; 棒10砖定位
KEEP(11) HR10.02  ; 棒11放砖至棒10
; rung 91: 棒10#过砖定位
LD 1.00  ; 棒10#光电
AND 101.11  ; 棒10#正转
TIM 011 #3
; rung 92: 棒10#放砖条件
LD 1.00  ; 棒10#光电
AND 2.11  ; 中线升降接近
ANDNOT 103.02  ; 中线升降
ANDNOT 100.12  ; 中线正转
ANDNOT 101.08  ; 棒8#
ANDNOT 101.09  ; 棍9#正转
ANDNOT 101.10  ; 棍9#反转
ANDNOT 0.15  ; 棒8#光电
ANDNOT 101.11  ; 棒10#正转
ANDNOT 101.12  ; 棒10#反转
ANDNOT 0.08  ; 连锁
TIM 042 #5
; rung 93: 棒8#放砖
LD TIM042  ; 棒10#放砖条件
LD CNT009  ; 棒10#放砖时间
KEEP(11) HR10.03  ; 棒10#放砖

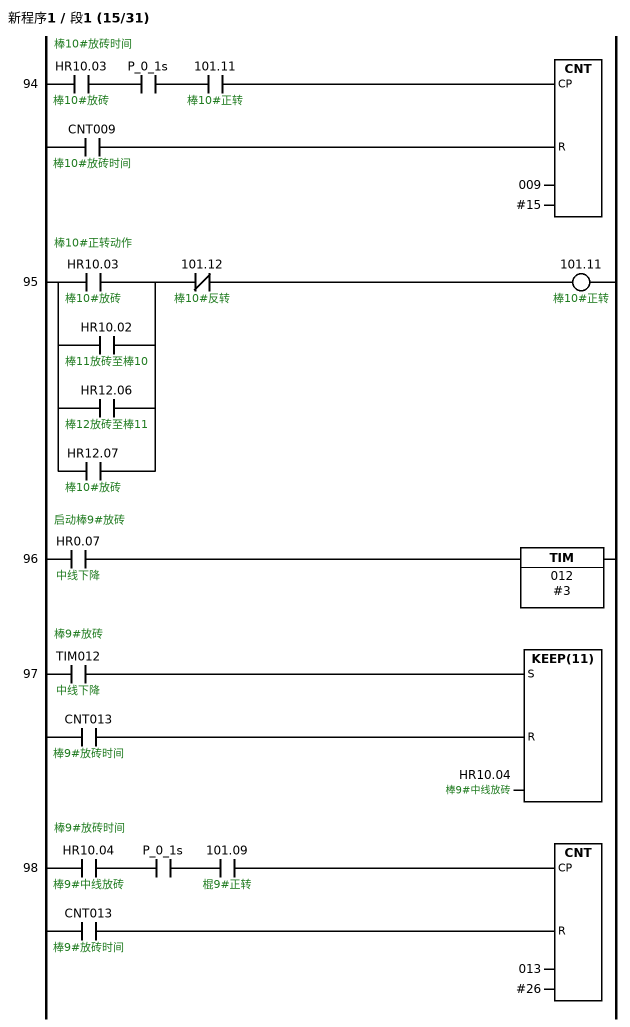
; rung 94: 棒10#放砖时间
LD HR10.03  ; 棒10#放砖
AND P_0_1s
AND 101.11  ; 棒10#正转
LD CNT009  ; 棒10#放砖时间
CNT 009 #15
; rung 95: 棒10#正转动作
LD HR10.03  ; 棒10#放砖
OR HR10.02  ; 棒11放砖至棒10
OR HR12.06  ; 棒12放砖至棒11
OR HR12.07  ; 棒10#放砖
ANDNOT 101.12  ; 棒10#反转
OUT 101.11  ; 棒10#正转
; rung 96: 启动棒9#放砖
LD HR0.07  ; 中线下降
TIM 012 #3
; rung 97: 棒9#放砖
LD TIM012  ; 中线下降
LD CNT013  ; 棒9#放砖时间
KEEP(11) HR10.04  ; 棒9#中线放砖
; rung 98: 棒9#放砖时间
LD HR10.04  ; 棒9#中线放砖
AND P_0_1s
AND 101.09  ; 棍9#正转
LD CNT013  ; 棒9#放砖时间
CNT 013 #26

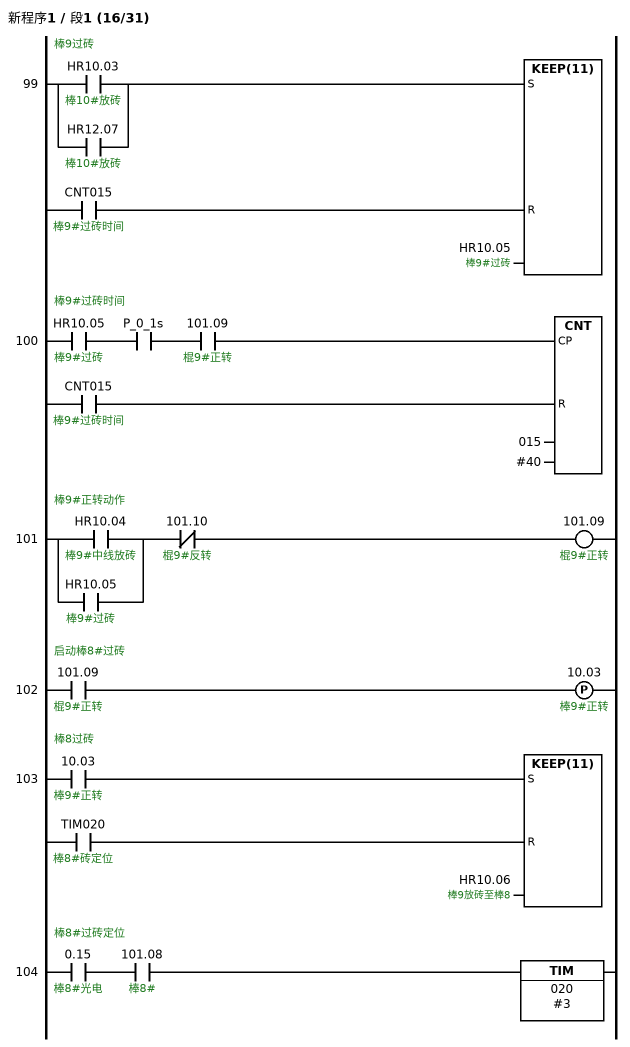
; rung 99: 棒9过砖
LD HR10.03  ; 棒10#放砖
OR HR12.07  ; 棒10#放砖
LD CNT015  ; 棒9#过砖时间
KEEP(11) HR10.05  ; 棒9#过砖
; rung 100: 棒9#过砖时间
LD HR10.05  ; 棒9#过砖
AND P_0_1s
AND 101.09  ; 棍9#正转
LD CNT015  ; 棒9#过砖时间
CNT 015 #40
; rung 101: 棒9#正转动作
LD HR10.04  ; 棒9#中线放砖
OR HR10.05  ; 棒9#过砖
ANDNOT 101.10  ; 棍9#反转
OUT 101.09  ; 棍9#正转
; rung 102: 启动棒8#过砖
LD 101.09  ; 棍9#正转
DIFU(13) 10.03  ; 棒9#正转
; rung 103: 棒8过砖
LD 10.03  ; 棒9#正转
LD TIM020  ; 棒8#砖定位
KEEP(11) HR10.06  ; 棒9放砖至棒8
; rung 104: 棒8#过砖定位
LD 0.15  ; 棒8#光电
AND 101.08  ; 棒8#
TIM 020 #3

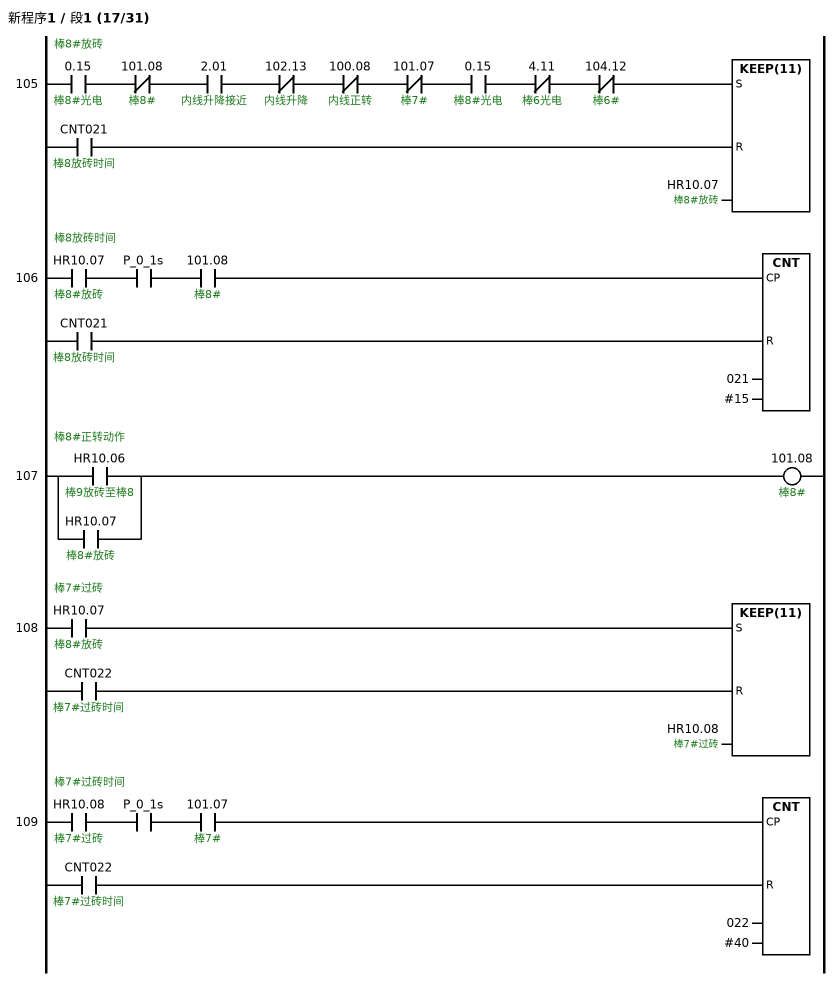
; rung 105: 棒8#放砖
LD 0.15  ; 棒8#光电
ANDNOT 101.08  ; 棒8#
AND 2.01  ; 内线升降接近
ANDNOT 102.13  ; 内线升降
ANDNOT 100.08  ; 内线正转
ANDNOT 101.07  ; 棒7#
AND 0.15  ; 棒8#光电
ANDNOT 4.11  ; 棒6光电
ANDNOT 104.12  ; 棒6#
LD CNT021  ; 棒8放砖时间
KEEP(11) HR10.07  ; 棒8#放砖
; rung 106: 棒8放砖时间
LD HR10.07  ; 棒8#放砖
AND P_0_1s
AND 101.08  ; 棒8#
LD CNT021  ; 棒8放砖时间
CNT 021 #15
; rung 107: 棒8#正转动作
LD HR10.06  ; 棒9放砖至棒8
OR HR10.07  ; 棒8#放砖
OUT 101.08  ; 棒8#
; rung 108: 棒7#过砖
LD HR10.07  ; 棒8#放砖
LD CNT022  ; 棒7#过砖时间
KEEP(11) HR10.08  ; 棒7#过砖
; rung 109: 棒7#过砖时间
LD HR10.08  ; 棒7#过砖
AND P_0_1s
AND 101.07  ; 棒7#
LD CNT022  ; 棒7#过砖时间
CNT 022 #40

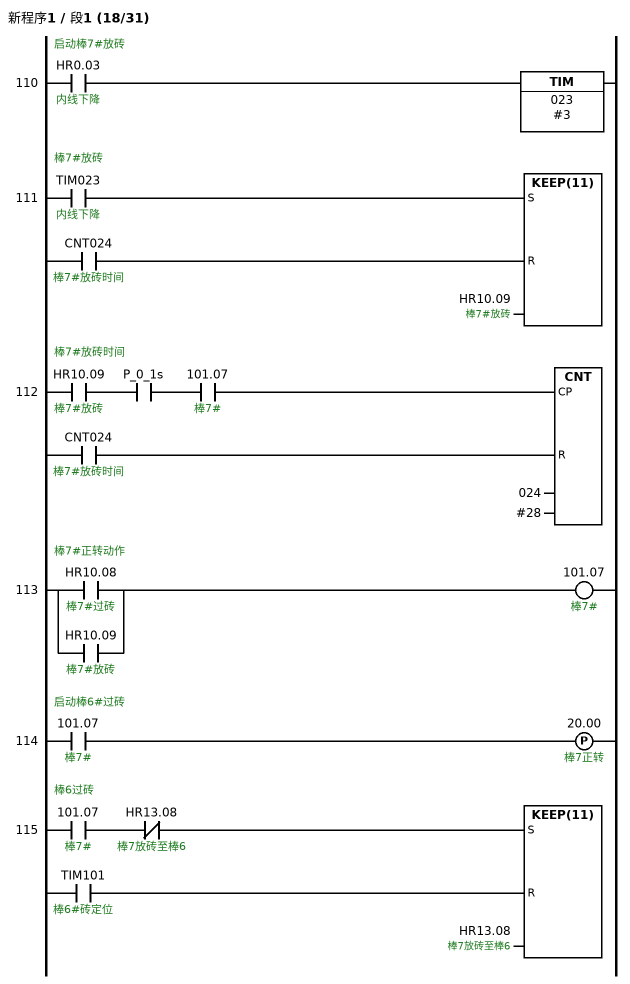
; rung 110: 启动棒7#放砖
LD HR0.03  ; 内线下降
TIM 023 #3
; rung 111: 棒7#放砖
LD TIM023  ; 内线下降
LD CNT024  ; 棒7#放砖时间
KEEP(11) HR10.09  ; 棒7#放砖
; rung 112: 棒7#放砖时间
LD HR10.09  ; 棒7#放砖
AND P_0_1s
AND 101.07  ; 棒7#
LD CNT024  ; 棒7#放砖时间
CNT 024 #28
; rung 113: 棒7#正转动作
LD HR10.08  ; 棒7#过砖
OR HR10.09  ; 棒7#放砖
OUT 101.07  ; 棒7#
; rung 114: 启动棒6#过砖
LD 101.07  ; 棒7#
DIFU(13) 20.00  ; 棒7正转
; rung 115: 棒6过砖
LD 101.07  ; 棒7#
ANDNOT HR13.08  ; 棒7放砖至棒6
LD TIM101  ; 棒6#砖定位
KEEP(11) HR13.08  ; 棒7放砖至棒6

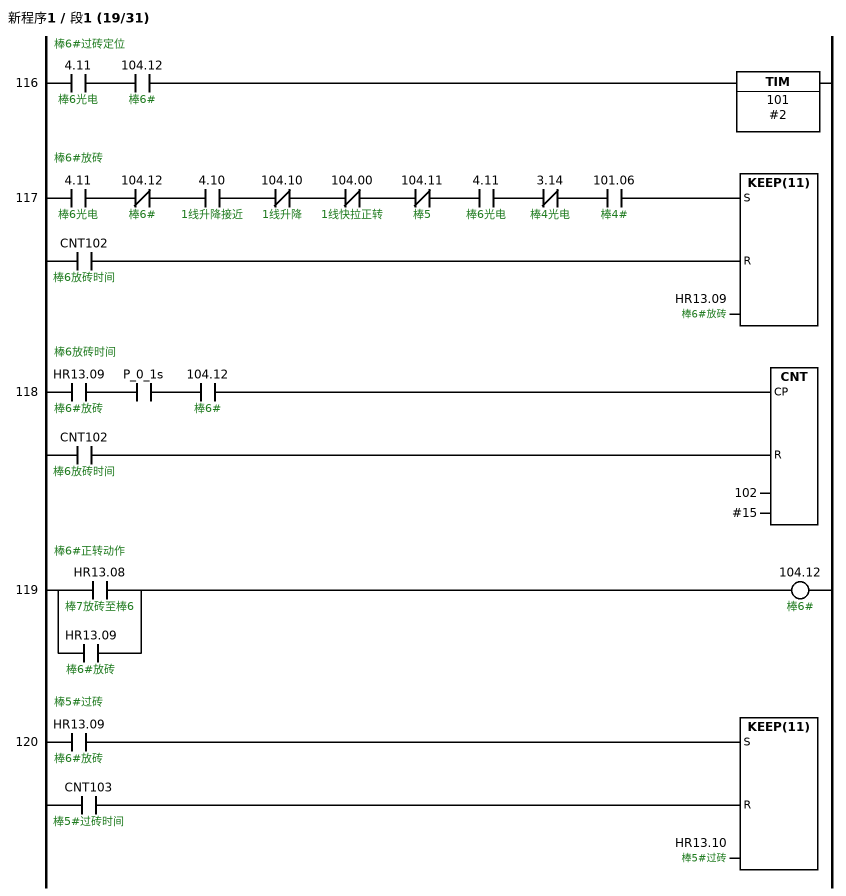
; rung 116: 棒6#过砖定位
LD 4.11  ; 棒6光电
AND 104.12  ; 棒6#
TIM 101 #2
; rung 117: 棒6#放砖
LD 4.11  ; 棒6光电
ANDNOT 104.12  ; 棒6#
AND 4.10  ; 1线升降接近
ANDNOT 104.10  ; 1线升降
ANDNOT 104.00  ; 1线快拉正转
ANDNOT 104.11  ; 棒5
AND 4.11  ; 棒6光电
ANDNOT 3.14  ; 棒4光电
AND 101.06  ; 棒4#
LD CNT102  ; 棒6放砖时间
KEEP(11) HR13.09  ; 棒6#放砖
; rung 118: 棒6放砖时间
LD HR13.09  ; 棒6#放砖
AND P_0_1s
AND 104.12  ; 棒6#
LD CNT102  ; 棒6放砖时间
CNT 102 #15
; rung 119: 棒6#正转动作
LD HR13.08  ; 棒7放砖至棒6
OR HR13.09  ; 棒6#放砖
OUT 104.12  ; 棒6#
; rung 120: 棒5#过砖
LD HR13.09  ; 棒6#放砖
LD CNT103  ; 棒5#过砖时间
KEEP(11) HR13.10  ; 棒5#过砖

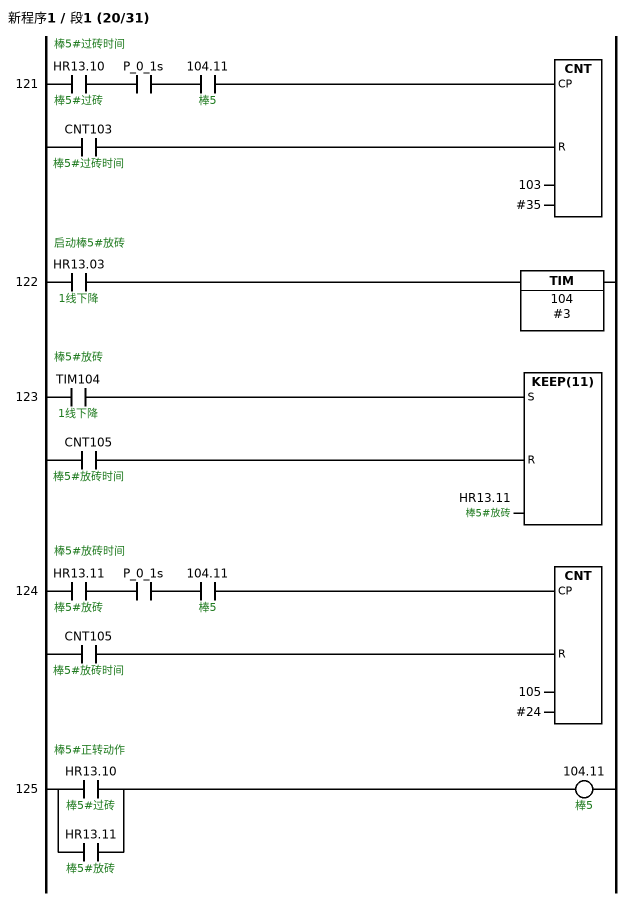
; rung 121: 棒5#过砖时间
LD HR13.10  ; 棒5#过砖
AND P_0_1s
AND 104.11  ; 棒5
LD CNT103  ; 棒5#过砖时间
CNT 103 #35
; rung 122: 启动棒5#放砖
LD HR13.03  ; 1线下降
TIM 104 #3
; rung 123: 棒5#放砖
LD TIM104  ; 1线下降
LD CNT105  ; 棒5#放砖时间
KEEP(11) HR13.11  ; 棒5#放砖
; rung 124: 棒5#放砖时间
LD HR13.11  ; 棒5#放砖
AND P_0_1s
AND 104.11  ; 棒5
LD CNT105  ; 棒5#放砖时间
CNT 105 #24
; rung 125: 棒5#正转动作
LD HR13.10  ; 棒5#过砖
OR HR13.11  ; 棒5#放砖
OUT 104.11  ; 棒5

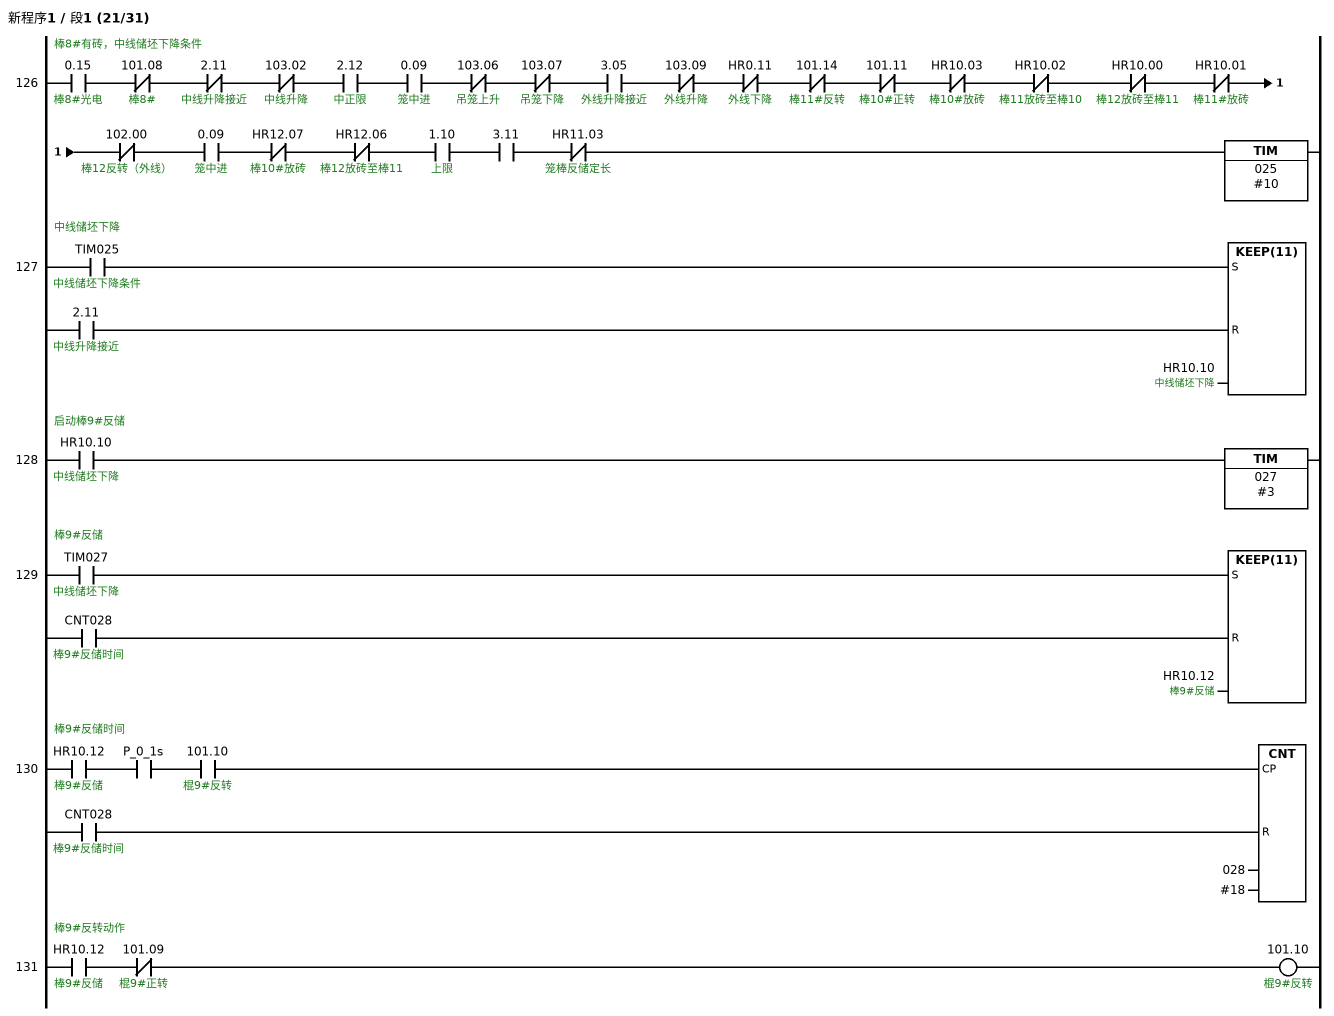
; rung 126: 棒8#有砖，中线储坯下降条件
LD 0.15  ; 棒8#光电
ANDNOT 101.08  ; 棒8#
ANDNOT 2.11  ; 中线升降接近
ANDNOT 103.02  ; 中线升降
AND 2.12  ; 中正限
AND 0.09  ; 笼中进
ANDNOT 103.06  ; 吊笼上升
ANDNOT 103.07  ; 吊笼下降
AND 3.05  ; 外线升降接近
ANDNOT 103.09  ; 外线升降
ANDNOT HR0.11  ; 外线下降
ANDNOT 101.14  ; 棒11#反转
ANDNOT 101.11  ; 棒10#正转
ANDNOT HR10.03  ; 棒10#放砖
ANDNOT HR10.02  ; 棒11放砖至棒10
ANDNOT HR10.00  ; 棒12放砖至棒11
ANDNOT HR10.01  ; 棒11#放砖
ANDNOT 102.00  ; 棒12反转（外线）
AND 0.09  ; 笼中进
ANDNOT HR12.07  ; 棒10#放砖
ANDNOT HR12.06  ; 棒12放砖至棒11
AND 1.10  ; 上限
AND 3.11
ANDNOT HR11.03  ; 笼棒反储定长
TIM 025 #10
; rung 127: 中线储坯下降
LD TIM025  ; 中线储坯下降条件
LD 2.11  ; 中线升降接近
KEEP(11) HR10.10  ; 中线储坯下降
; rung 128: 启动棒9#反储
LD HR10.10  ; 中线储坯下降
TIM 027 #3
; rung 129: 棒9#反储
LD TIM027  ; 中线储坯下降
LD CNT028  ; 棒9#反储时间
KEEP(11) HR10.12  ; 棒9#反储
; rung 130: 棒9#反储时间
LD HR10.12  ; 棒9#反储
AND P_0_1s
AND 101.10  ; 棍9#反转
LD CNT028  ; 棒9#反储时间
CNT 028 #18
; rung 131: 棒9#反转动作
LD HR10.12  ; 棒9#反储
ANDNOT 101.09  ; 棍9#正转
OUT 101.10  ; 棍9#反转

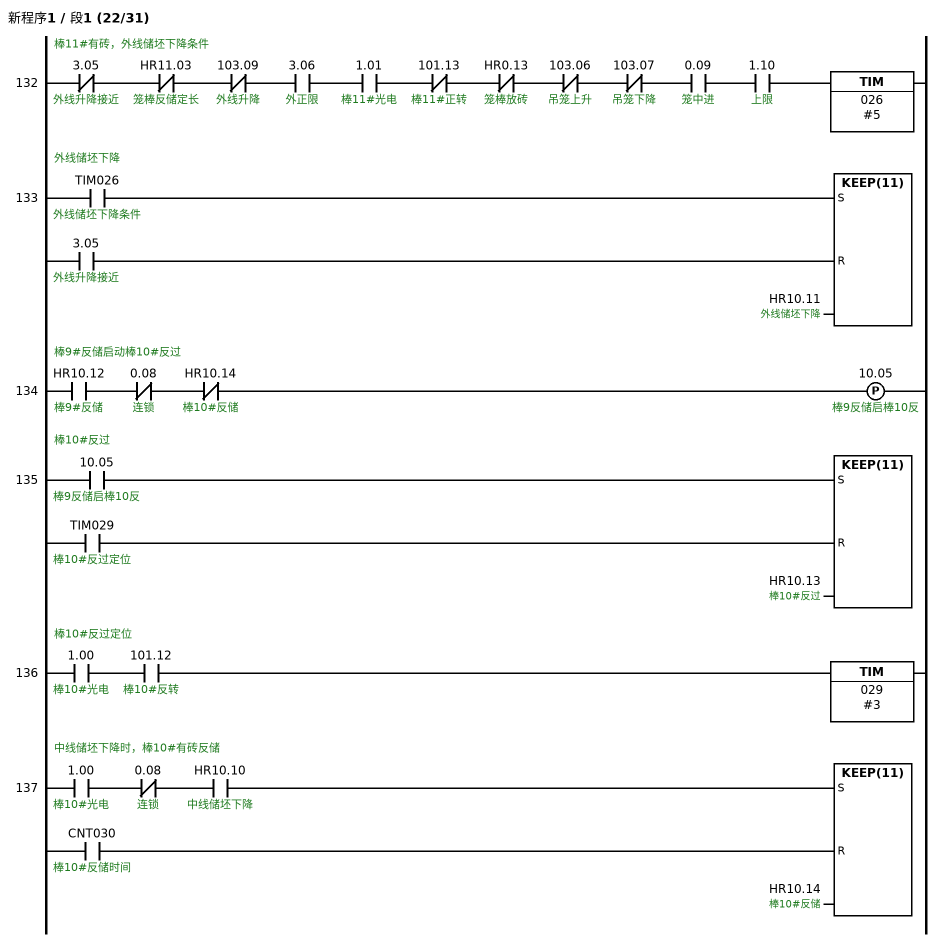
; rung 132: 棒11#有砖，外线储坯下降条件
LDNOT 3.05  ; 外线升降接近
ANDNOT HR11.03  ; 笼棒反储定长
ANDNOT 103.09  ; 外线升降
AND 3.06  ; 外正限
AND 1.01  ; 棒11#光电
ANDNOT 101.13  ; 棒11#正转
ANDNOT HR0.13  ; 笼棒放砖
ANDNOT 103.06  ; 吊笼上升
ANDNOT 103.07  ; 吊笼下降
AND 0.09  ; 笼中进
AND 1.10  ; 上限
TIM 026 #5
; rung 133: 外线储坯下降
LD TIM026  ; 外线储坯下降条件
LD 3.05  ; 外线升降接近
KEEP(11) HR10.11  ; 外线储坯下降
; rung 134: 棒9#反储启动棒10#反过
LD HR10.12  ; 棒9#反储
ANDNOT 0.08  ; 连锁
ANDNOT HR10.14  ; 棒10#反储
DIFU(13) 10.05  ; 棒9反储启棒10反
; rung 135: 棒10#反过
LD 10.05  ; 棒9反储启棒10反
LD TIM029  ; 棒10#反过定位
KEEP(11) HR10.13  ; 棒10#反过
; rung 136: 棒10#反过定位
LD 1.00  ; 棒10#光电
AND 101.12  ; 棒10#反转
TIM 029 #3
; rung 137: 中线储坯下降时，棒10#有砖反储
LD 1.00  ; 棒10#光电
ANDNOT 0.08  ; 连锁
AND HR10.10  ; 中线储坯下降
LD CNT030  ; 棒10#反储时间
KEEP(11) HR10.14  ; 棒10#反储

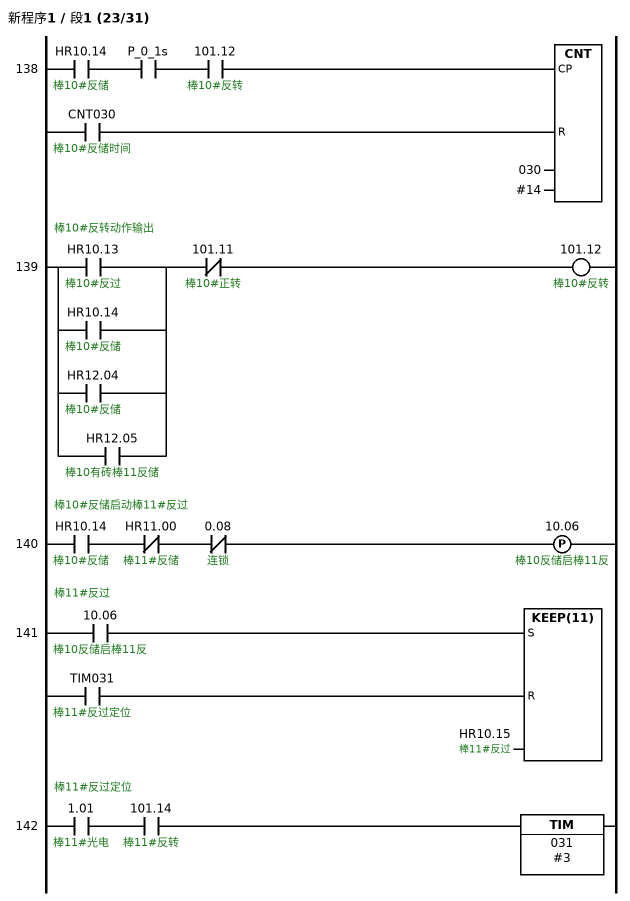
; rung 138
LD HR10.14  ; 棒10#反储
AND P_0_1s
AND 101.12  ; 棒10#反转
LD CNT030  ; 棒10#反储时间
CNT 030 #14
; rung 139: 棒10#反转动作输出
LD HR10.13  ; 棒10#反过
OR HR10.14  ; 棒10#反储
OR HR12.04  ; 棒10#反储
OR HR12.05  ; 棒10有砖棒11反储
ANDNOT 101.11  ; 棒10#正转
OUT 101.12  ; 棒10#反转
; rung 140: 棒10#反储启动棒11#反过
LD HR10.14  ; 棒10#反储
ANDNOT HR11.00  ; 棒11#反储
ANDNOT 0.08  ; 连锁
DIFU(13) 10.06  ; 棒10反储启棒11反
; rung 141: 棒11#反过
LD 10.06  ; 棒10反储启棒11反
LD TIM031  ; 棒11#反过定位
KEEP(11) HR10.15  ; 棒11#反过
; rung 142: 棒11#反过定位
LD 1.01  ; 棒11#光电
AND 101.14  ; 棒11#反转
TIM 031 #3

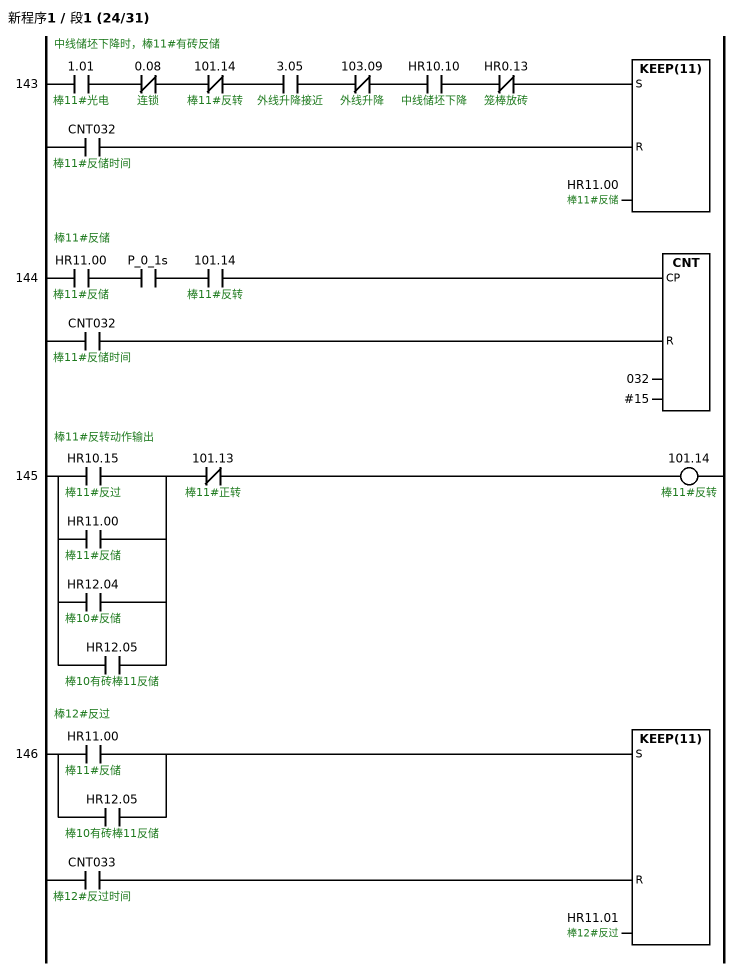
; rung 143: 中线储坯下降时，棒11#有砖反储
LD 1.01  ; 棒11#光电
ANDNOT 0.08  ; 连锁
ANDNOT 101.14  ; 棒11#反转
AND 3.05  ; 外线升降接近
ANDNOT 103.09  ; 外线升降
AND HR10.10  ; 中线储坯下降
ANDNOT HR0.13  ; 笼棒放砖
LD CNT032  ; 棒11#反储时间
KEEP(11) HR11.00  ; 棒11#反储
; rung 144: 棒11#反储
LD HR11.00  ; 棒11#反储
AND P_0_1s
AND 101.14  ; 棒11#反转
LD CNT032  ; 棒11#反储时间
CNT 032 #15
; rung 145: 棒11#反转动作输出
LD HR10.15  ; 棒11#反过
OR HR11.00  ; 棒11#反储
OR HR12.04  ; 棒10#反储
OR HR12.05  ; 棒10有砖棒11反储
ANDNOT 101.13  ; 棒11#正转
OUT 101.14  ; 棒11#反转
; rung 146: 棒12#反过
LD HR11.00  ; 棒11#反储
OR HR12.05  ; 棒10有砖棒11反储
LD CNT033  ; 棒12#反过时间
KEEP(11) HR11.01  ; 棒12#反过

